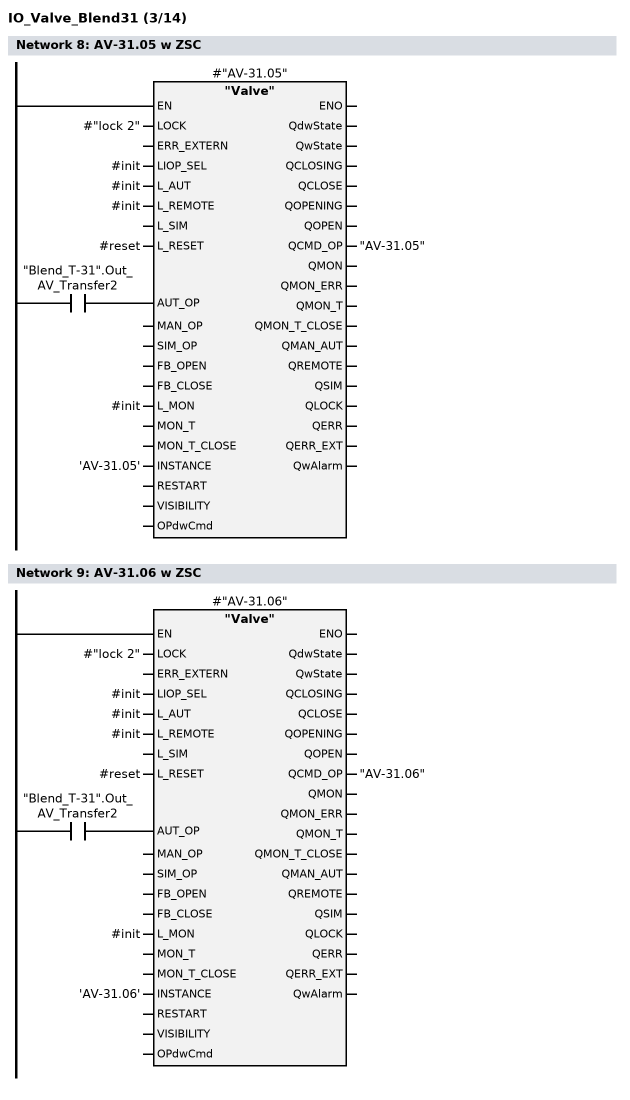
   RUNG wire#powerrail
      #"AV-31.05"(AUT_OP := wire#w1, LOCK := #"lock 2", ERR_EXTERN :=, LIOP_SEL := #init, L_AUT := #init, L_REMOTE := #init, L_SIM :=, L_RESET := #reset, MAN_OP :=, SIM_OP :=, FB_OPEN :=, FB_CLOSE :=, L_MON := #init, MON_T :=, MON_T_CLOSE :=, INSTANCE := 'AV-31.05', RESTART :=, VISIBILITY :=, OPdwCmd :=, QdwState =>, QwState =>, QCLOSING =>, QCLOSE =>, QOPENING =>, QOPEN =>, QCMD_OP => "AV-31.05", QMON =>, QMON_ERR =>, QMON_T =>, QMON_T_CLOSE =>, QMAN_AUT =>, QREMOTE =>, QSIM =>, QLOCK =>, QERR =>, QERR_EXT =>, QwAlarm =>)
   END_RUNG
   RUNG wire#powerrail
      Contact( "Blend_T-31".Out_AV_Transfer2 )
   END_RUNG wire#w1
   // the same network as SCL:
   #"AV-31.05"(LOCK := #"lock 2",   // "Valve"
               LIOP_SEL := #init,
               L_AUT := #init,
               L_REMOTE := #init,
               L_RESET := #reset,
               AUT_OP := "Blend_T-31".Out_AV_Transfer2,
               L_MON := #init,
               INSTANCE := 'AV-31.05',
               QCMD_OP => "AV-31.05");
END_REGION

REGION Network 9: AV-31.06 w ZSC
   RUNG wire#powerrail
      #"AV-31.06"(AUT_OP := wire#w1, LOCK := #"lock 2", ERR_EXTERN :=, LIOP_SEL := #init, L_AUT := #init, L_REMOTE := #init, L_SIM :=, L_RESET := #reset, MAN_OP :=, SIM_OP :=, FB_OPEN :=, FB_CLOSE :=, L_MON := #init, MON_T :=, MON_T_CLOSE :=, INSTANCE := 'AV-31.06', RESTART :=, VISIBILITY :=, OPdwCmd :=, QdwState =>, QwState =>, QCLOSING =>, QCLOSE =>, QOPENING =>, QOPEN =>, QCMD_OP => "AV-31.06", QMON =>, QMON_ERR =>, QMON_T =>, QMON_T_CLOSE =>, QMAN_AUT =>, QREMOTE =>, QSIM =>, QLOCK =>, QERR =>, QERR_EXT =>, QwAlarm =>)
   END_RUNG
   RUNG wire#powerrail
      Contact( "Blend_T-31".Out_AV_Transfer2 )
   END_RUNG wire#w1
   // the same network as SCL:
   #"AV-31.06"(LOCK := #"lock 2",   // "Valve"
               LIOP_SEL := #init,
               L_AUT := #init,
               L_REMOTE := #init,
               L_RESET := #reset,
               AUT_OP := "Blend_T-31".Out_AV_Transfer2,
               L_MON := #init,
               INSTANCE := 'AV-31.06',
               QCMD_OP => "AV-31.06");
END_REGION

REGION Network 10: AV-31.07
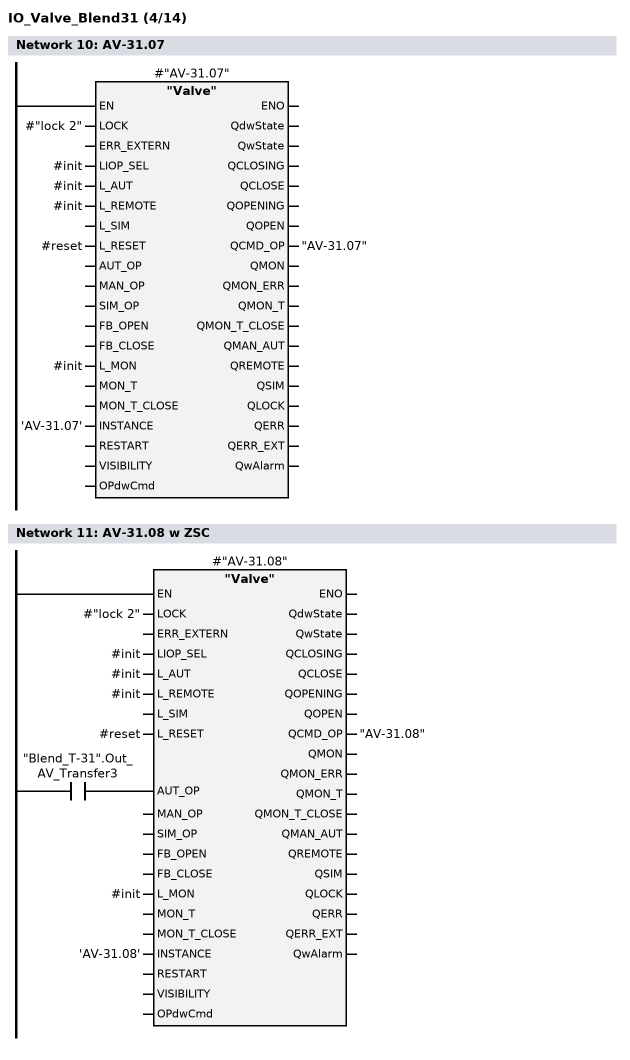
   RUNG wire#powerrail
      #"AV-31.07"(LOCK := #"lock 2", ERR_EXTERN :=, LIOP_SEL := #init, L_AUT := #init, L_REMOTE := #init, L_SIM :=, L_RESET := #reset, AUT_OP :=, MAN_OP :=, SIM_OP :=, FB_OPEN :=, FB_CLOSE :=, L_MON := #init, MON_T :=, MON_T_CLOSE :=, INSTANCE := 'AV-31.07', RESTART :=, VISIBILITY :=, OPdwCmd :=, QdwState =>, QwState =>, QCLOSING =>, QCLOSE =>, QOPENING =>, QOPEN =>, QCMD_OP => "AV-31.07", QMON =>, QMON_ERR =>, QMON_T =>, QMON_T_CLOSE =>, QMAN_AUT =>, QREMOTE =>, QSIM =>, QLOCK =>, QERR =>, QERR_EXT =>, QwAlarm =>)
   END_RUNG
   // the same network as SCL:
   #"AV-31.07"(LOCK := #"lock 2",   // "Valve"
               LIOP_SEL := #init,
               L_AUT := #init,
               L_REMOTE := #init,
               L_RESET := #reset,
               L_MON := #init,
               INSTANCE := 'AV-31.07',
               QCMD_OP => "AV-31.07");
END_REGION

REGION Network 11: AV-31.08 w ZSC
   RUNG wire#powerrail
      #"AV-31.08"(AUT_OP := wire#w1, LOCK := #"lock 2", ERR_EXTERN :=, LIOP_SEL := #init, L_AUT := #init, L_REMOTE := #init, L_SIM :=, L_RESET := #reset, MAN_OP :=, SIM_OP :=, FB_OPEN :=, FB_CLOSE :=, L_MON := #init, MON_T :=, MON_T_CLOSE :=, INSTANCE := 'AV-31.08', RESTART :=, VISIBILITY :=, OPdwCmd :=, QdwState =>, QwState =>, QCLOSING =>, QCLOSE =>, QOPENING =>, QOPEN =>, QCMD_OP => "AV-31.08", QMON =>, QMON_ERR =>, QMON_T =>, QMON_T_CLOSE =>, QMAN_AUT =>, QREMOTE =>, QSIM =>, QLOCK =>, QERR =>, QERR_EXT =>, QwAlarm =>)
   END_RUNG
   RUNG wire#powerrail
      Contact( "Blend_T-31".Out_AV_Transfer3 )
   END_RUNG wire#w1
   // the same network as SCL:
   #"AV-31.08"(LOCK := #"lock 2",   // "Valve"
               LIOP_SEL := #init,
               L_AUT := #init,
               L_REMOTE := #init,
               L_RESET := #reset,
               AUT_OP := "Blend_T-31".Out_AV_Transfer3,
               L_MON := #init,
               INSTANCE := 'AV-31.08',
               QCMD_OP => "AV-31.08");
END_REGION

REGION Network 12: AV-31.09 w ZSC
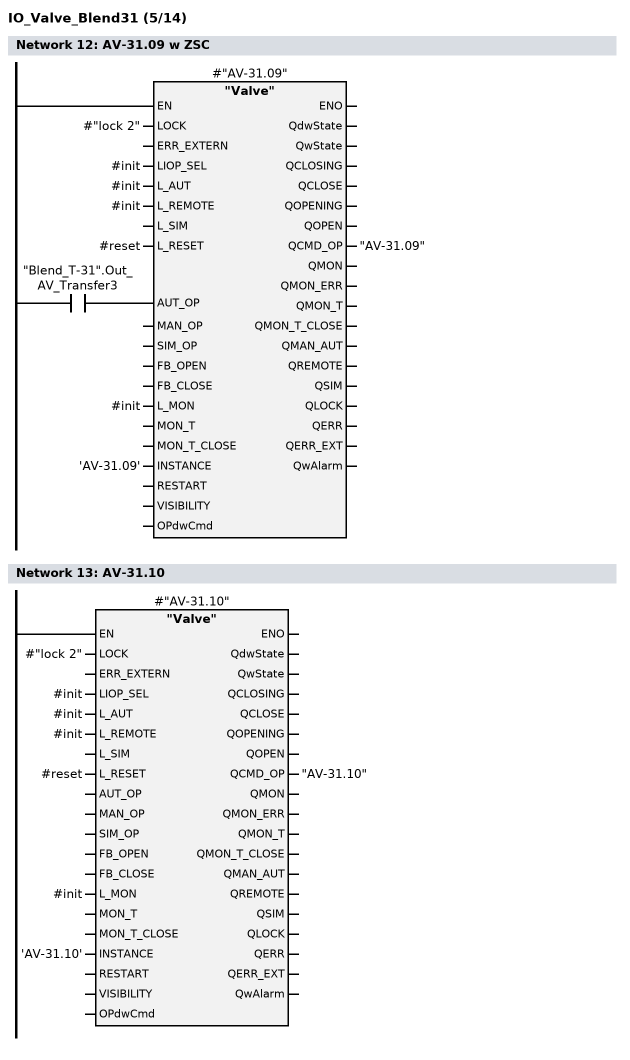
   RUNG wire#powerrail
      #"AV-31.09"(AUT_OP := wire#w1, LOCK := #"lock 2", ERR_EXTERN :=, LIOP_SEL := #init, L_AUT := #init, L_REMOTE := #init, L_SIM :=, L_RESET := #reset, MAN_OP :=, SIM_OP :=, FB_OPEN :=, FB_CLOSE :=, L_MON := #init, MON_T :=, MON_T_CLOSE :=, INSTANCE := 'AV-31.09', RESTART :=, VISIBILITY :=, OPdwCmd :=, QdwState =>, QwState =>, QCLOSING =>, QCLOSE =>, QOPENING =>, QOPEN =>, QCMD_OP => "AV-31.09", QMON =>, QMON_ERR =>, QMON_T =>, QMON_T_CLOSE =>, QMAN_AUT =>, QREMOTE =>, QSIM =>, QLOCK =>, QERR =>, QERR_EXT =>, QwAlarm =>)
   END_RUNG
   RUNG wire#powerrail
      Contact( "Blend_T-31".Out_AV_Transfer3 )
   END_RUNG wire#w1
   // the same network as SCL:
   #"AV-31.09"(LOCK := #"lock 2",   // "Valve"
               LIOP_SEL := #init,
               L_AUT := #init,
               L_REMOTE := #init,
               L_RESET := #reset,
               AUT_OP := "Blend_T-31".Out_AV_Transfer3,
               L_MON := #init,
               INSTANCE := 'AV-31.09',
               QCMD_OP => "AV-31.09");
END_REGION

REGION Network 13: AV-31.10
   RUNG wire#powerrail
      #"AV-31.10"(LOCK := #"lock 2", ERR_EXTERN :=, LIOP_SEL := #init, L_AUT := #init, L_REMOTE := #init, L_SIM :=, L_RESET := #reset, AUT_OP :=, MAN_OP :=, SIM_OP :=, FB_OPEN :=, FB_CLOSE :=, L_MON := #init, MON_T :=, MON_T_CLOSE :=, INSTANCE := 'AV-31.10', RESTART :=, VISIBILITY :=, OPdwCmd :=, QdwState =>, QwState =>, QCLOSING =>, QCLOSE =>, QOPENING =>, QOPEN =>, QCMD_OP => "AV-31.10", QMON =>, QMON_ERR =>, QMON_T =>, QMON_T_CLOSE =>, QMAN_AUT =>, QREMOTE =>, QSIM =>, QLOCK =>, QERR =>, QERR_EXT =>, QwAlarm =>)
   END_RUNG
   // the same network as SCL:
   #"AV-31.10"(LOCK := #"lock 2",   // "Valve"
               LIOP_SEL := #init,
               L_AUT := #init,
               L_REMOTE := #init,
               L_RESET := #reset,
               L_MON := #init,
               INSTANCE := 'AV-31.10',
               QCMD_OP => "AV-31.10");
END_REGION

REGION Network 14: AV-31.11 w ZSC
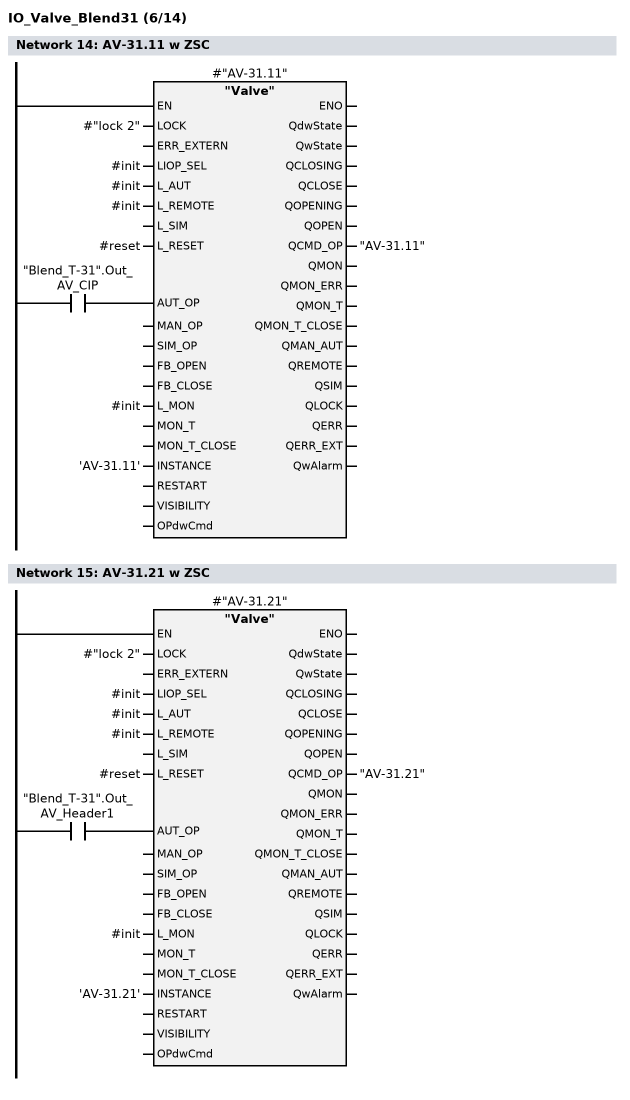
   RUNG wire#powerrail
      #"AV-31.11"(AUT_OP := wire#w1, LOCK := #"lock 2", ERR_EXTERN :=, LIOP_SEL := #init, L_AUT := #init, L_REMOTE := #init, L_SIM :=, L_RESET := #reset, MAN_OP :=, SIM_OP :=, FB_OPEN :=, FB_CLOSE :=, L_MON := #init, MON_T :=, MON_T_CLOSE :=, INSTANCE := 'AV-31.11', RESTART :=, VISIBILITY :=, OPdwCmd :=, QdwState =>, QwState =>, QCLOSING =>, QCLOSE =>, QOPENING =>, QOPEN =>, QCMD_OP => "AV-31.11", QMON =>, QMON_ERR =>, QMON_T =>, QMON_T_CLOSE =>, QMAN_AUT =>, QREMOTE =>, QSIM =>, QLOCK =>, QERR =>, QERR_EXT =>, QwAlarm =>)
   END_RUNG
   RUNG wire#powerrail
      Contact( "Blend_T-31".Out_AV_CIP )
   END_RUNG wire#w1
   // the same network as SCL:
   #"AV-31.11"(LOCK := #"lock 2",   // "Valve"
               LIOP_SEL := #init,
               L_AUT := #init,
               L_REMOTE := #init,
               L_RESET := #reset,
               AUT_OP := "Blend_T-31".Out_AV_CIP,
               L_MON := #init,
               INSTANCE := 'AV-31.11',
               QCMD_OP => "AV-31.11");
END_REGION

REGION Network 15: AV-31.21 w ZSC
   RUNG wire#powerrail
      #"AV-31.21"(AUT_OP := wire#w1, LOCK := #"lock 2", ERR_EXTERN :=, LIOP_SEL := #init, L_AUT := #init, L_REMOTE := #init, L_SIM :=, L_RESET := #reset, MAN_OP :=, SIM_OP :=, FB_OPEN :=, FB_CLOSE :=, L_MON := #init, MON_T :=, MON_T_CLOSE :=, INSTANCE := 'AV-31.21', RESTART :=, VISIBILITY :=, OPdwCmd :=, QdwState =>, QwState =>, QCLOSING =>, QCLOSE =>, QOPENING =>, QOPEN =>, QCMD_OP => "AV-31.21", QMON =>, QMON_ERR =>, QMON_T =>, QMON_T_CLOSE =>, QMAN_AUT =>, QREMOTE =>, QSIM =>, QLOCK =>, QERR =>, QERR_EXT =>, QwAlarm =>)
   END_RUNG
   RUNG wire#powerrail
      Contact( "Blend_T-31".Out_AV_Header1 )
   END_RUNG wire#w1
   // the same network as SCL:
   #"AV-31.21"(LOCK := #"lock 2",   // "Valve"
               LIOP_SEL := #init,
               L_AUT := #init,
               L_REMOTE := #init,
               L_RESET := #reset,
               AUT_OP := "Blend_T-31".Out_AV_Header1,
               L_MON := #init,
               INSTANCE := 'AV-31.21',
               QCMD_OP => "AV-31.21");
END_REGION

REGION Network 16: AV-31.22
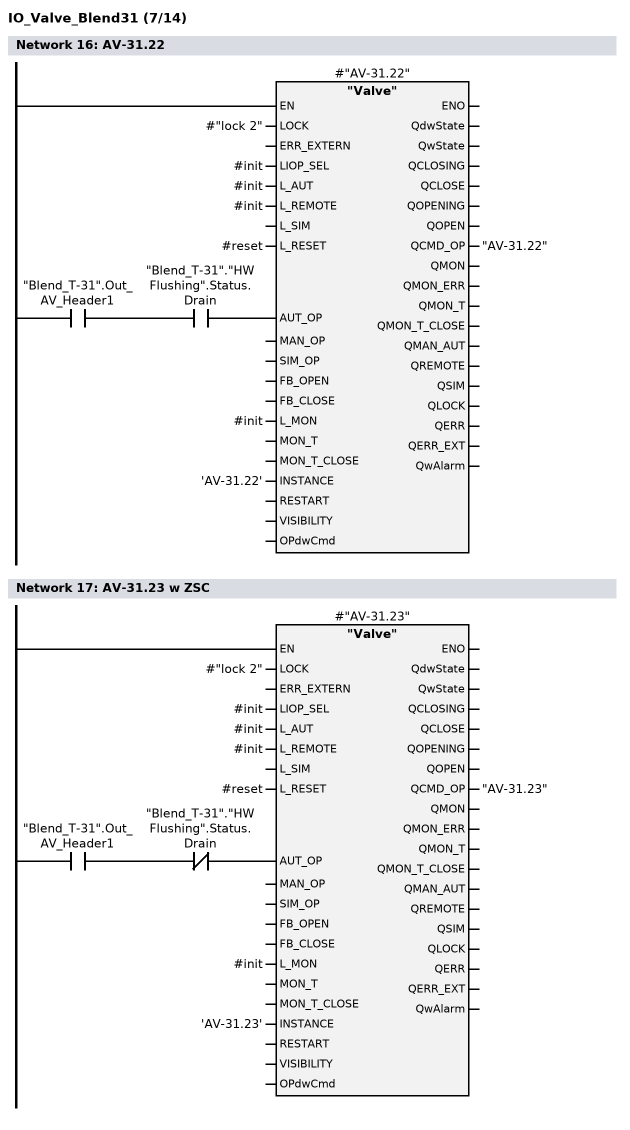
   RUNG wire#powerrail
      #"AV-31.22"(AUT_OP := wire#w1, LOCK := #"lock 2", ERR_EXTERN :=, LIOP_SEL := #init, L_AUT := #init, L_REMOTE := #init, L_SIM :=, L_RESET := #reset, MAN_OP :=, SIM_OP :=, FB_OPEN :=, FB_CLOSE :=, L_MON := #init, MON_T :=, MON_T_CLOSE :=, INSTANCE := 'AV-31.22', RESTART :=, VISIBILITY :=, OPdwCmd :=, QdwState =>, QwState =>, QCLOSING =>, QCLOSE =>, QOPENING =>, QOPEN =>, QCMD_OP => "AV-31.22", QMON =>, QMON_ERR =>, QMON_T =>, QMON_T_CLOSE =>, QMAN_AUT =>, QREMOTE =>, QSIM =>, QLOCK =>, QERR =>, QERR_EXT =>, QwAlarm =>)
   END_RUNG
   RUNG wire#powerrail
      Contact( "Blend_T-31".Out_AV_Header1 )
      Contact( "Blend_T-31"."HW Flushing".Status.Drain )
   END_RUNG wire#w1
   // the same network as SCL:
   #"AV-31.22"(LOCK := #"lock 2",   // "Valve"
               LIOP_SEL := #init,
               L_AUT := #init,
               L_REMOTE := #init,
               L_RESET := #reset,
               AUT_OP := "Blend_T-31".Out_AV_Header1 AND "Blend_T-31"."HW Flushing".Status.Drain,
               L_MON := #init,
               INSTANCE := 'AV-31.22',
               QCMD_OP => "AV-31.22");
END_REGION

REGION Network 17: AV-31.23 w ZSC
   RUNG wire#powerrail
      #"AV-31.23"(AUT_OP := wire#w1, LOCK := #"lock 2", ERR_EXTERN :=, LIOP_SEL := #init, L_AUT := #init, L_REMOTE := #init, L_SIM :=, L_RESET := #reset, MAN_OP :=, SIM_OP :=, FB_OPEN :=, FB_CLOSE :=, L_MON := #init, MON_T :=, MON_T_CLOSE :=, INSTANCE := 'AV-31.23', RESTART :=, VISIBILITY :=, OPdwCmd :=, QdwState =>, QwState =>, QCLOSING =>, QCLOSE =>, QOPENING =>, QOPEN =>, QCMD_OP => "AV-31.23", QMON =>, QMON_ERR =>, QMON_T =>, QMON_T_CLOSE =>, QMAN_AUT =>, QREMOTE =>, QSIM =>, QLOCK =>, QERR =>, QERR_EXT =>, QwAlarm =>)
   END_RUNG
   RUNG wire#powerrail
      Contact( "Blend_T-31".Out_AV_Header1 )
      I_Contact( "Blend_T-31"."HW Flushing".Status.Drain )
   END_RUNG wire#w1
   // the same network as SCL:
   #"AV-31.23"(LOCK := #"lock 2",   // "Valve"
               LIOP_SEL := #init,
               L_AUT := #init,
               L_REMOTE := #init,
               L_RESET := #reset,
               AUT_OP := "Blend_T-31".Out_AV_Header1 AND NOT "Blend_T-31"."HW Flushing".Status.Drain,
               L_MON := #init,
               INSTANCE := 'AV-31.23',
               QCMD_OP => "AV-31.23");
END_REGION

REGION Network 18: AV-31.24 w ZSC
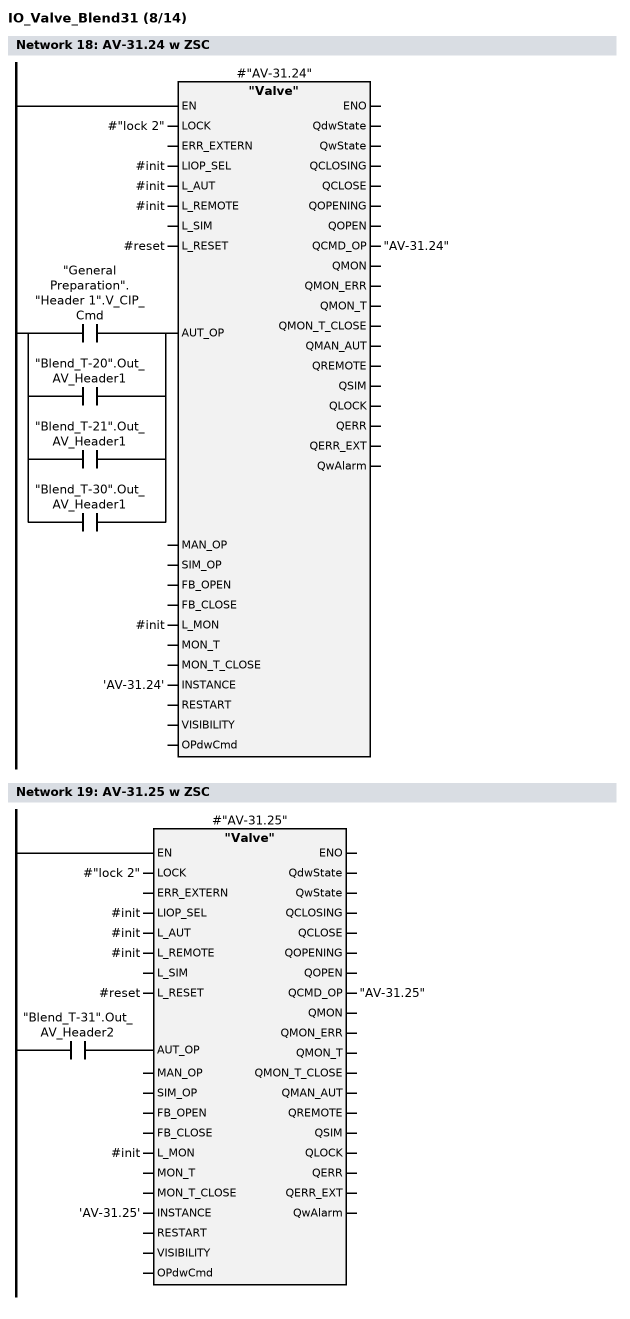
   RUNG wire#powerrail
      #"AV-31.24"(AUT_OP := wire#w1, LOCK := #"lock 2", ERR_EXTERN :=, LIOP_SEL := #init, L_AUT := #init, L_REMOTE := #init, L_SIM :=, L_RESET := #reset, MAN_OP :=, SIM_OP :=, FB_OPEN :=, FB_CLOSE :=, L_MON := #init, MON_T :=, MON_T_CLOSE :=, INSTANCE := 'AV-31.24', RESTART :=, VISIBILITY :=, OPdwCmd :=, QdwState =>, QwState =>, QCLOSING =>, QCLOSE =>, QOPENING =>, QOPEN =>, QCMD_OP => "AV-31.24", QMON =>, QMON_ERR =>, QMON_T =>, QMON_T_CLOSE =>, QMAN_AUT =>, QREMOTE =>, QSIM =>, QLOCK =>, QERR =>, QERR_EXT =>, QwAlarm =>)
   END_RUNG
   RUNG wire#powerrail
      Contact( "General Preparation"."Header 1".V_CIP_Cmd )
   END_RUNG wire#w1
   RUNG wire#powerrail
      Contact( "Blend_T-20".Out_AV_Header1 )
   END_RUNG wire#w1
   RUNG wire#powerrail
      Contact( "Blend_T-21".Out_AV_Header1 )
   END_RUNG wire#w1
   RUNG wire#powerrail
      Contact( "Blend_T-30".Out_AV_Header1 )
   END_RUNG wire#w1
   // the same network as SCL:
   #"AV-31.24"(LOCK := #"lock 2",   // "Valve"
               LIOP_SEL := #init,
               L_AUT := #init,
               L_REMOTE := #init,
               L_RESET := #reset,
               AUT_OP := "General Preparation"."Header 1".V_CIP_Cmd OR "Blend_T-20".Out_AV_Header1 OR "Blend_T-21".Out_AV_Header1 OR "Blend_T-30".Out_AV_Header1,
               L_MON := #init,
               INSTANCE := 'AV-31.24',
               QCMD_OP => "AV-31.24");
END_REGION

REGION Network 19: AV-31.25 w ZSC
   RUNG wire#powerrail
      #"AV-31.25"(AUT_OP := wire#w1, LOCK := #"lock 2", ERR_EXTERN :=, LIOP_SEL := #init, L_AUT := #init, L_REMOTE := #init, L_SIM :=, L_RESET := #reset, MAN_OP :=, SIM_OP :=, FB_OPEN :=, FB_CLOSE :=, L_MON := #init, MON_T :=, MON_T_CLOSE :=, INSTANCE := 'AV-31.25', RESTART :=, VISIBILITY :=, OPdwCmd :=, QdwState =>, QwState =>, QCLOSING =>, QCLOSE =>, QOPENING =>, QOPEN =>, QCMD_OP => "AV-31.25", QMON =>, QMON_ERR =>, QMON_T =>, QMON_T_CLOSE =>, QMAN_AUT =>, QREMOTE =>, QSIM =>, QLOCK =>, QERR =>, QERR_EXT =>, QwAlarm =>)
   END_RUNG
   RUNG wire#powerrail
      Contact( "Blend_T-31".Out_AV_Header2 )
   END_RUNG wire#w1
   // the same network as SCL:
   #"AV-31.25"(LOCK := #"lock 2",   // "Valve"
               LIOP_SEL := #init,
               L_AUT := #init,
               L_REMOTE := #init,
               L_RESET := #reset,
               AUT_OP := "Blend_T-31".Out_AV_Header2,
               L_MON := #init,
               INSTANCE := 'AV-31.25',
               QCMD_OP => "AV-31.25");
END_REGION

REGION Network 20: AV-31.26
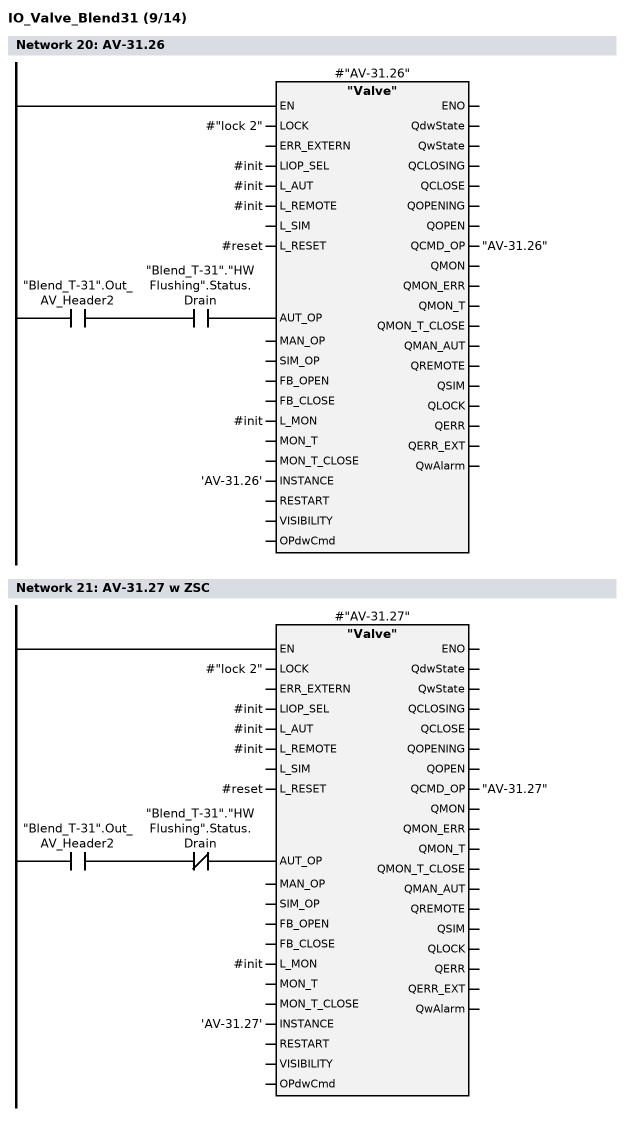
   RUNG wire#powerrail
      #"AV-31.26"(AUT_OP := wire#w1, LOCK := #"lock 2", ERR_EXTERN :=, LIOP_SEL := #init, L_AUT := #init, L_REMOTE := #init, L_SIM :=, L_RESET := #reset, MAN_OP :=, SIM_OP :=, FB_OPEN :=, FB_CLOSE :=, L_MON := #init, MON_T :=, MON_T_CLOSE :=, INSTANCE := 'AV-31.26', RESTART :=, VISIBILITY :=, OPdwCmd :=, QdwState =>, QwState =>, QCLOSING =>, QCLOSE =>, QOPENING =>, QOPEN =>, QCMD_OP => "AV-31.26", QMON =>, QMON_ERR =>, QMON_T =>, QMON_T_CLOSE =>, QMAN_AUT =>, QREMOTE =>, QSIM =>, QLOCK =>, QERR =>, QERR_EXT =>, QwAlarm =>)
   END_RUNG
   RUNG wire#powerrail
      Contact( "Blend_T-31".Out_AV_Header2 )
      Contact( "Blend_T-31"."HW Flushing".Status.Drain )
   END_RUNG wire#w1
   // the same network as SCL:
   #"AV-31.26"(LOCK := #"lock 2",   // "Valve"
               LIOP_SEL := #init,
               L_AUT := #init,
               L_REMOTE := #init,
               L_RESET := #reset,
               AUT_OP := "Blend_T-31".Out_AV_Header2 AND "Blend_T-31"."HW Flushing".Status.Drain,
               L_MON := #init,
               INSTANCE := 'AV-31.26',
               QCMD_OP => "AV-31.26");
END_REGION

REGION Network 21: AV-31.27 w ZSC
   RUNG wire#powerrail
      #"AV-31.27"(AUT_OP := wire#w1, LOCK := #"lock 2", ERR_EXTERN :=, LIOP_SEL := #init, L_AUT := #init, L_REMOTE := #init, L_SIM :=, L_RESET := #reset, MAN_OP :=, SIM_OP :=, FB_OPEN :=, FB_CLOSE :=, L_MON := #init, MON_T :=, MON_T_CLOSE :=, INSTANCE := 'AV-31.27', RESTART :=, VISIBILITY :=, OPdwCmd :=, QdwState =>, QwState =>, QCLOSING =>, QCLOSE =>, QOPENING =>, QOPEN =>, QCMD_OP => "AV-31.27", QMON =>, QMON_ERR =>, QMON_T =>, QMON_T_CLOSE =>, QMAN_AUT =>, QREMOTE =>, QSIM =>, QLOCK =>, QERR =>, QERR_EXT =>, QwAlarm =>)
   END_RUNG
   RUNG wire#powerrail
      Contact( "Blend_T-31".Out_AV_Header2 )
      I_Contact( "Blend_T-31"."HW Flushing".Status.Drain )
   END_RUNG wire#w1
   // the same network as SCL:
   #"AV-31.27"(LOCK := #"lock 2",   // "Valve"
               LIOP_SEL := #init,
               L_AUT := #init,
               L_REMOTE := #init,
               L_RESET := #reset,
               AUT_OP := "Blend_T-31".Out_AV_Header2 AND NOT "Blend_T-31"."HW Flushing".Status.Drain,
               L_MON := #init,
               INSTANCE := 'AV-31.27',
               QCMD_OP => "AV-31.27");
END_REGION

REGION Network 22: AV-31.28 w ZSC
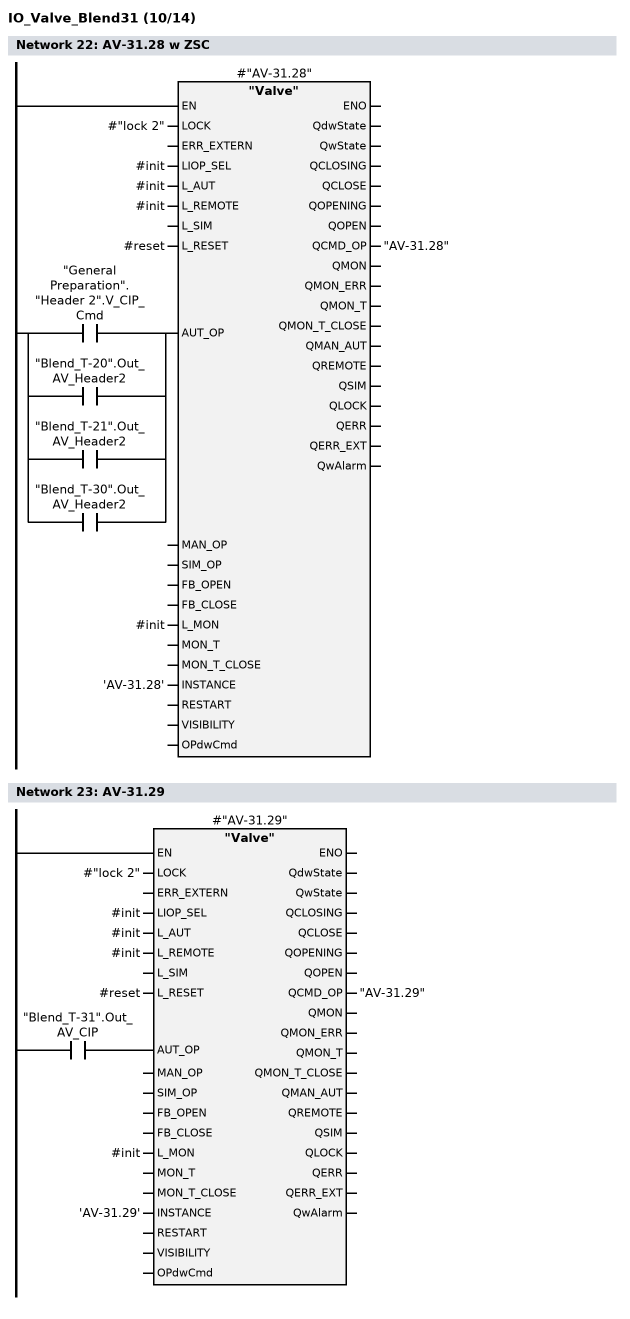
   RUNG wire#powerrail
      #"AV-31.28"(AUT_OP := wire#w1, LOCK := #"lock 2", ERR_EXTERN :=, LIOP_SEL := #init, L_AUT := #init, L_REMOTE := #init, L_SIM :=, L_RESET := #reset, MAN_OP :=, SIM_OP :=, FB_OPEN :=, FB_CLOSE :=, L_MON := #init, MON_T :=, MON_T_CLOSE :=, INSTANCE := 'AV-31.28', RESTART :=, VISIBILITY :=, OPdwCmd :=, QdwState =>, QwState =>, QCLOSING =>, QCLOSE =>, QOPENING =>, QOPEN =>, QCMD_OP => "AV-31.28", QMON =>, QMON_ERR =>, QMON_T =>, QMON_T_CLOSE =>, QMAN_AUT =>, QREMOTE =>, QSIM =>, QLOCK =>, QERR =>, QERR_EXT =>, QwAlarm =>)
   END_RUNG
   RUNG wire#powerrail
      Contact( "General Preparation"."Header 2".V_CIP_Cmd )
   END_RUNG wire#w1
   RUNG wire#powerrail
      Contact( "Blend_T-20".Out_AV_Header2 )
   END_RUNG wire#w1
   RUNG wire#powerrail
      Contact( "Blend_T-21".Out_AV_Header2 )
   END_RUNG wire#w1
   RUNG wire#powerrail
      Contact( "Blend_T-30".Out_AV_Header2 )
   END_RUNG wire#w1
   // the same network as SCL:
   #"AV-31.28"(LOCK := #"lock 2",   // "Valve"
               LIOP_SEL := #init,
               L_AUT := #init,
               L_REMOTE := #init,
               L_RESET := #reset,
               AUT_OP := "General Preparation"."Header 2".V_CIP_Cmd OR "Blend_T-20".Out_AV_Header2 OR "Blend_T-21".Out_AV_Header2 OR "Blend_T-30".Out_AV_Header2,
               L_MON := #init,
               INSTANCE := 'AV-31.28',
               QCMD_OP => "AV-31.28");
END_REGION

REGION Network 23: AV-31.29
   RUNG wire#powerrail
      #"AV-31.29"(AUT_OP := wire#w1, LOCK := #"lock 2", ERR_EXTERN :=, LIOP_SEL := #init, L_AUT := #init, L_REMOTE := #init, L_SIM :=, L_RESET := #reset, MAN_OP :=, SIM_OP :=, FB_OPEN :=, FB_CLOSE :=, L_MON := #init, MON_T :=, MON_T_CLOSE :=, INSTANCE := 'AV-31.29', RESTART :=, VISIBILITY :=, OPdwCmd :=, QdwState =>, QwState =>, QCLOSING =>, QCLOSE =>, QOPENING =>, QOPEN =>, QCMD_OP => "AV-31.29", QMON =>, QMON_ERR =>, QMON_T =>, QMON_T_CLOSE =>, QMAN_AUT =>, QREMOTE =>, QSIM =>, QLOCK =>, QERR =>, QERR_EXT =>, QwAlarm =>)
   END_RUNG
   RUNG wire#powerrail
      Contact( "Blend_T-31".Out_AV_CIP )
   END_RUNG wire#w1
   // the same network as SCL:
   #"AV-31.29"(LOCK := #"lock 2",   // "Valve"
               LIOP_SEL := #init,
               L_AUT := #init,
               L_REMOTE := #init,
               L_RESET := #reset,
               AUT_OP := "Blend_T-31".Out_AV_CIP,
               L_MON := #init,
               INSTANCE := 'AV-31.29',
               QCMD_OP => "AV-31.29");
END_REGION

REGION Network 24: AV-31.30
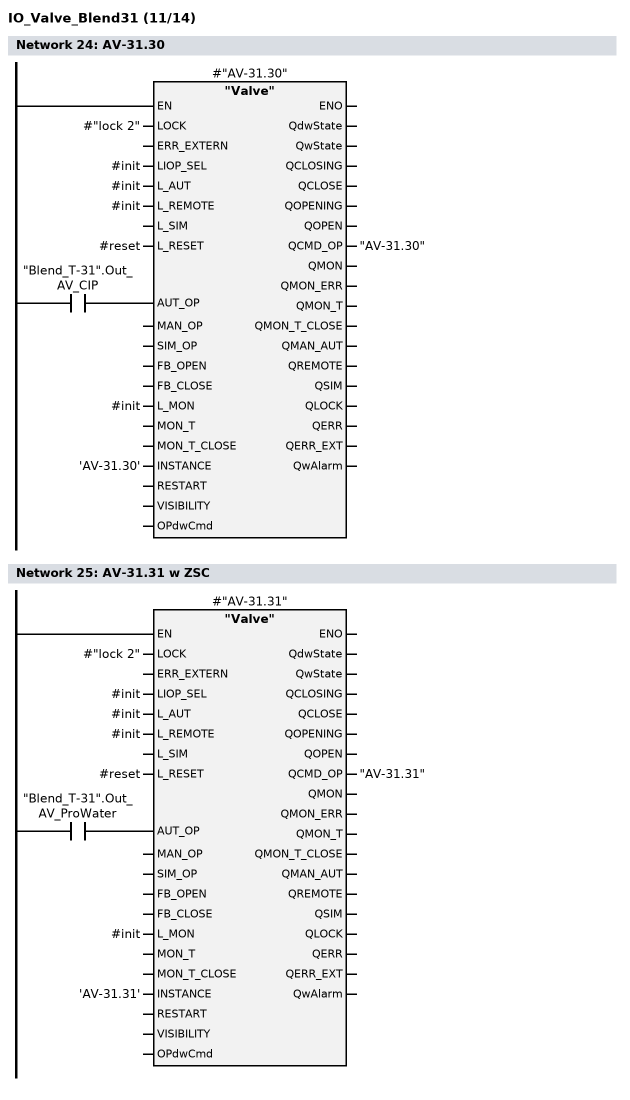
   RUNG wire#powerrail
      #"AV-31.30"(AUT_OP := wire#w1, LOCK := #"lock 2", ERR_EXTERN :=, LIOP_SEL := #init, L_AUT := #init, L_REMOTE := #init, L_SIM :=, L_RESET := #reset, MAN_OP :=, SIM_OP :=, FB_OPEN :=, FB_CLOSE :=, L_MON := #init, MON_T :=, MON_T_CLOSE :=, INSTANCE := 'AV-31.30', RESTART :=, VISIBILITY :=, OPdwCmd :=, QdwState =>, QwState =>, QCLOSING =>, QCLOSE =>, QOPENING =>, QOPEN =>, QCMD_OP => "AV-31.30", QMON =>, QMON_ERR =>, QMON_T =>, QMON_T_CLOSE =>, QMAN_AUT =>, QREMOTE =>, QSIM =>, QLOCK =>, QERR =>, QERR_EXT =>, QwAlarm =>)
   END_RUNG
   RUNG wire#powerrail
      Contact( "Blend_T-31".Out_AV_CIP )
   END_RUNG wire#w1
   // the same network as SCL:
   #"AV-31.30"(LOCK := #"lock 2",   // "Valve"
               LIOP_SEL := #init,
               L_AUT := #init,
               L_REMOTE := #init,
               L_RESET := #reset,
               AUT_OP := "Blend_T-31".Out_AV_CIP,
               L_MON := #init,
               INSTANCE := 'AV-31.30',
               QCMD_OP => "AV-31.30");
END_REGION

REGION Network 25: AV-31.31 w ZSC
   RUNG wire#powerrail
      #"AV-31.31"(AUT_OP := wire#w1, LOCK := #"lock 2", ERR_EXTERN :=, LIOP_SEL := #init, L_AUT := #init, L_REMOTE := #init, L_SIM :=, L_RESET := #reset, MAN_OP :=, SIM_OP :=, FB_OPEN :=, FB_CLOSE :=, L_MON := #init, MON_T :=, MON_T_CLOSE :=, INSTANCE := 'AV-31.31', RESTART :=, VISIBILITY :=, OPdwCmd :=, QdwState =>, QwState =>, QCLOSING =>, QCLOSE =>, QOPENING =>, QOPEN =>, QCMD_OP => "AV-31.31", QMON =>, QMON_ERR =>, QMON_T =>, QMON_T_CLOSE =>, QMAN_AUT =>, QREMOTE =>, QSIM =>, QLOCK =>, QERR =>, QERR_EXT =>, QwAlarm =>)
   END_RUNG
   RUNG wire#powerrail
      Contact( "Blend_T-31".Out_AV_ProWater )
   END_RUNG wire#w1
   // the same network as SCL:
   #"AV-31.31"(LOCK := #"lock 2",   // "Valve"
               LIOP_SEL := #init,
               L_AUT := #init,
               L_REMOTE := #init,
               L_RESET := #reset,
               AUT_OP := "Blend_T-31".Out_AV_ProWater,
               L_MON := #init,
               INSTANCE := 'AV-31.31',
               QCMD_OP => "AV-31.31");
END_REGION

REGION Network 26: AV-31.32 w ZSC
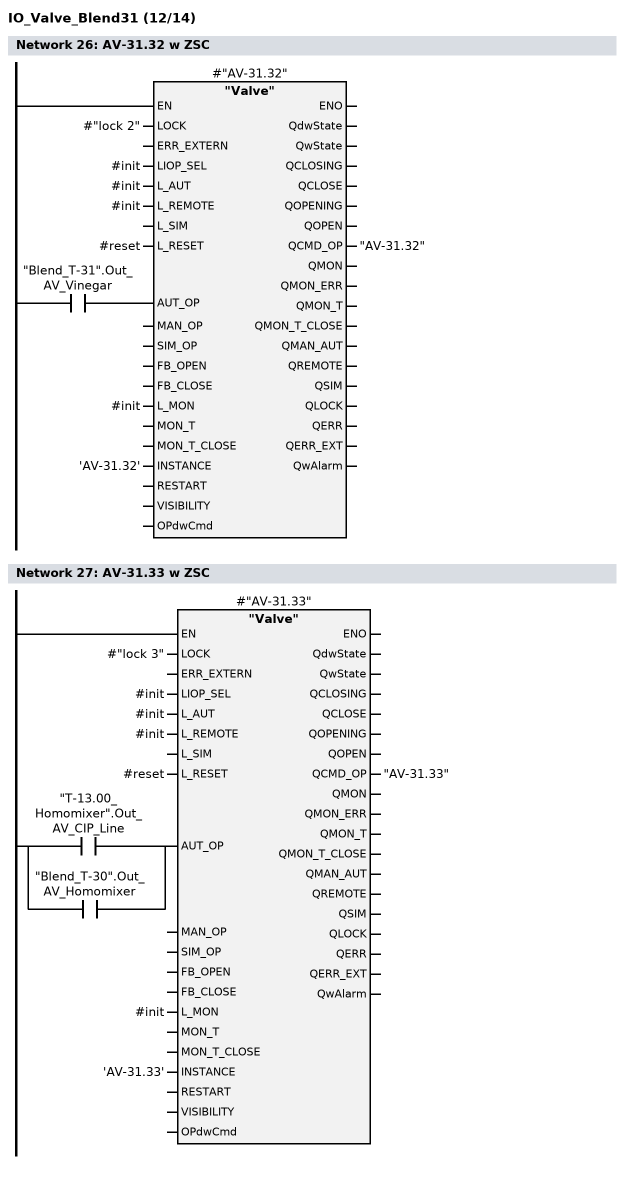
   RUNG wire#powerrail
      #"AV-31.32"(AUT_OP := wire#w1, LOCK := #"lock 2", ERR_EXTERN :=, LIOP_SEL := #init, L_AUT := #init, L_REMOTE := #init, L_SIM :=, L_RESET := #reset, MAN_OP :=, SIM_OP :=, FB_OPEN :=, FB_CLOSE :=, L_MON := #init, MON_T :=, MON_T_CLOSE :=, INSTANCE := 'AV-31.32', RESTART :=, VISIBILITY :=, OPdwCmd :=, QdwState =>, QwState =>, QCLOSING =>, QCLOSE =>, QOPENING =>, QOPEN =>, QCMD_OP => "AV-31.32", QMON =>, QMON_ERR =>, QMON_T =>, QMON_T_CLOSE =>, QMAN_AUT =>, QREMOTE =>, QSIM =>, QLOCK =>, QERR =>, QERR_EXT =>, QwAlarm =>)
   END_RUNG
   RUNG wire#powerrail
      Contact( "Blend_T-31".Out_AV_Vinegar )
   END_RUNG wire#w1
   // the same network as SCL:
   #"AV-31.32"(LOCK := #"lock 2",   // "Valve"
               LIOP_SEL := #init,
               L_AUT := #init,
               L_REMOTE := #init,
               L_RESET := #reset,
               AUT_OP := "Blend_T-31".Out_AV_Vinegar,
               L_MON := #init,
               INSTANCE := 'AV-31.32',
               QCMD_OP => "AV-31.32");
END_REGION

REGION Network 27: AV-31.33 w ZSC
   RUNG wire#powerrail
      #"AV-31.33"(AUT_OP := wire#w1, LOCK := #"lock 3", ERR_EXTERN :=, LIOP_SEL := #init, L_AUT := #init, L_REMOTE := #init, L_SIM :=, L_RESET := #reset, MAN_OP :=, SIM_OP :=, FB_OPEN :=, FB_CLOSE :=, L_MON := #init, MON_T :=, MON_T_CLOSE :=, INSTANCE := 'AV-31.33', RESTART :=, VISIBILITY :=, OPdwCmd :=, QdwState =>, QwState =>, QCLOSING =>, QCLOSE =>, QOPENING =>, QOPEN =>, QCMD_OP => "AV-31.33", QMON =>, QMON_ERR =>, QMON_T =>, QMON_T_CLOSE =>, QMAN_AUT =>, QREMOTE =>, QSIM =>, QLOCK =>, QERR =>, QERR_EXT =>, QwAlarm =>)
   END_RUNG
   RUNG wire#powerrail
      Contact( "T-13.00_Homomixer".Out_AV_CIP_Line )
   END_RUNG wire#w1
   RUNG wire#powerrail
      Contact( "Blend_T-30".Out_AV_Homomixer )
   END_RUNG wire#w1
   // the same network as SCL:
   #"AV-31.33"(LOCK := #"lock 3",   // "Valve"
               LIOP_SEL := #init,
               L_AUT := #init,
               L_REMOTE := #init,
               L_RESET := #reset,
               AUT_OP := "T-13.00_Homomixer".Out_AV_CIP_Line OR "Blend_T-30".Out_AV_Homomixer,
               L_MON := #init,
               INSTANCE := 'AV-31.33',
               QCMD_OP => "AV-31.33");
END_REGION

REGION Network 28: AV-31.34 w ZSC
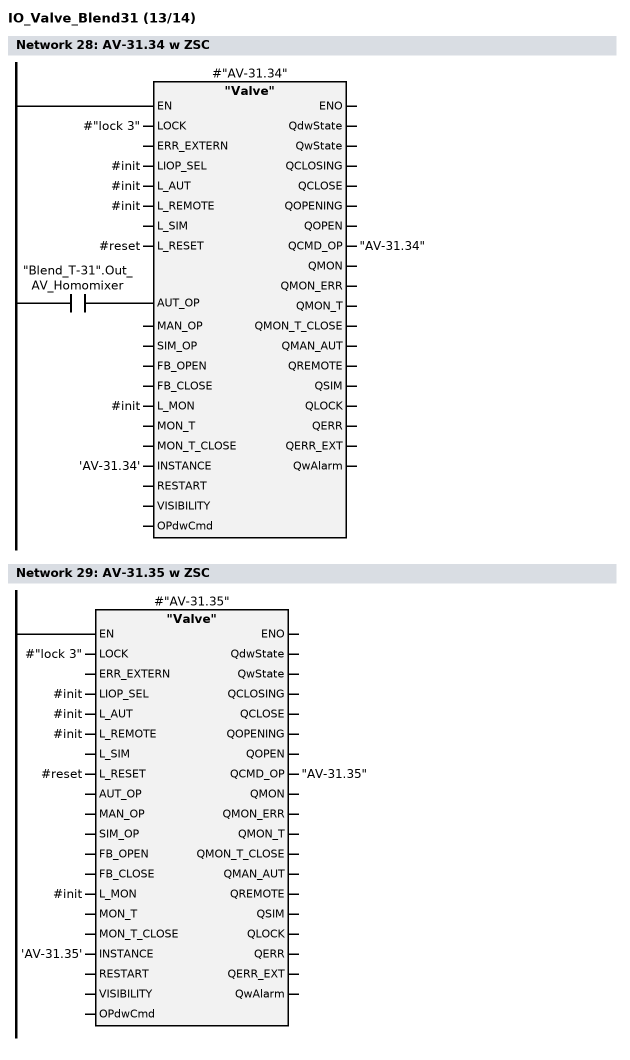
   RUNG wire#powerrail
      #"AV-31.34"(AUT_OP := wire#w1, LOCK := #"lock 3", ERR_EXTERN :=, LIOP_SEL := #init, L_AUT := #init, L_REMOTE := #init, L_SIM :=, L_RESET := #reset, MAN_OP :=, SIM_OP :=, FB_OPEN :=, FB_CLOSE :=, L_MON := #init, MON_T :=, MON_T_CLOSE :=, INSTANCE := 'AV-31.34', RESTART :=, VISIBILITY :=, OPdwCmd :=, QdwState =>, QwState =>, QCLOSING =>, QCLOSE =>, QOPENING =>, QOPEN =>, QCMD_OP => "AV-31.34", QMON =>, QMON_ERR =>, QMON_T =>, QMON_T_CLOSE =>, QMAN_AUT =>, QREMOTE =>, QSIM =>, QLOCK =>, QERR =>, QERR_EXT =>, QwAlarm =>)
   END_RUNG
   RUNG wire#powerrail
      Contact( "Blend_T-31".Out_AV_Homomixer )
   END_RUNG wire#w1
   // the same network as SCL:
   #"AV-31.34"(LOCK := #"lock 3",   // "Valve"
               LIOP_SEL := #init,
               L_AUT := #init,
               L_REMOTE := #init,
               L_RESET := #reset,
               AUT_OP := "Blend_T-31".Out_AV_Homomixer,
               L_MON := #init,
               INSTANCE := 'AV-31.34',
               QCMD_OP => "AV-31.34");
END_REGION

REGION Network 29: AV-31.35 w ZSC
   RUNG wire#powerrail
      #"AV-31.35"(LOCK := #"lock 3", ERR_EXTERN :=, LIOP_SEL := #init, L_AUT := #init, L_REMOTE := #init, L_SIM :=, L_RESET := #reset, AUT_OP :=, MAN_OP :=, SIM_OP :=, FB_OPEN :=, FB_CLOSE :=, L_MON := #init, MON_T :=, MON_T_CLOSE :=, INSTANCE := 'AV-31.35', RESTART :=, VISIBILITY :=, OPdwCmd :=, QdwState =>, QwState =>, QCLOSING =>, QCLOSE =>, QOPENING =>, QOPEN =>, QCMD_OP => "AV-31.35", QMON =>, QMON_ERR =>, QMON_T =>, QMON_T_CLOSE =>, QMAN_AUT =>, QREMOTE =>, QSIM =>, QLOCK =>, QERR =>, QERR_EXT =>, QwAlarm =>)
   END_RUNG
   // the same network as SCL:
   #"AV-31.35"(LOCK := #"lock 3",   // "Valve"
               LIOP_SEL := #init,
               L_AUT := #init,
               L_REMOTE := #init,
               L_RESET := #reset,
               L_MON := #init,
               INSTANCE := 'AV-31.35',
               QCMD_OP => "AV-31.35");
END_REGION

REGION Network 30: AV-31.41
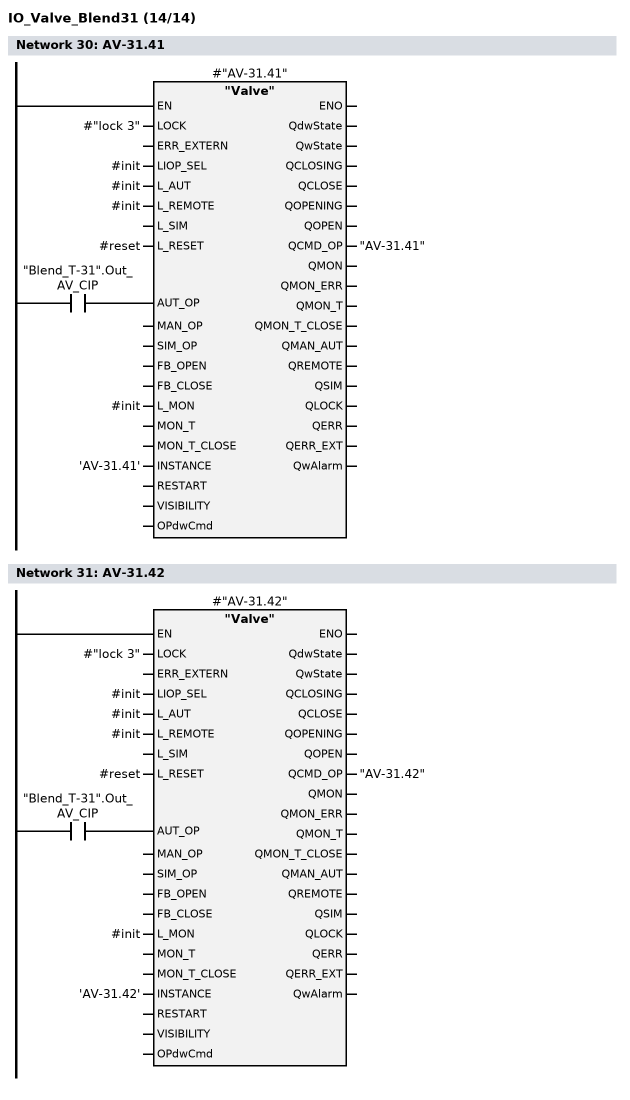
   RUNG wire#powerrail
      #"AV-31.41"(AUT_OP := wire#w1, LOCK := #"lock 3", ERR_EXTERN :=, LIOP_SEL := #init, L_AUT := #init, L_REMOTE := #init, L_SIM :=, L_RESET := #reset, MAN_OP :=, SIM_OP :=, FB_OPEN :=, FB_CLOSE :=, L_MON := #init, MON_T :=, MON_T_CLOSE :=, INSTANCE := 'AV-31.41', RESTART :=, VISIBILITY :=, OPdwCmd :=, QdwState =>, QwState =>, QCLOSING =>, QCLOSE =>, QOPENING =>, QOPEN =>, QCMD_OP => "AV-31.41", QMON =>, QMON_ERR =>, QMON_T =>, QMON_T_CLOSE =>, QMAN_AUT =>, QREMOTE =>, QSIM =>, QLOCK =>, QERR =>, QERR_EXT =>, QwAlarm =>)
   END_RUNG
   RUNG wire#powerrail
      Contact( "Blend_T-31".Out_AV_CIP )
   END_RUNG wire#w1
   // the same network as SCL:
   #"AV-31.41"(LOCK := #"lock 3",   // "Valve"
               LIOP_SEL := #init,
               L_AUT := #init,
               L_REMOTE := #init,
               L_RESET := #reset,
               AUT_OP := "Blend_T-31".Out_AV_CIP,
               L_MON := #init,
               INSTANCE := 'AV-31.41',
               QCMD_OP => "AV-31.41");
END_REGION

REGION Network 31: AV-31.42
   RUNG wire#powerrail
      #"AV-31.42"(AUT_OP := wire#w1, LOCK := #"lock 3", ERR_EXTERN :=, LIOP_SEL := #init, L_AUT := #init, L_REMOTE := #init, L_SIM :=, L_RESET := #reset, MAN_OP :=, SIM_OP :=, FB_OPEN :=, FB_CLOSE :=, L_MON := #init, MON_T :=, MON_T_CLOSE :=, INSTANCE := 'AV-31.42', RESTART :=, VISIBILITY :=, OPdwCmd :=, QdwState =>, QwState =>, QCLOSING =>, QCLOSE =>, QOPENING =>, QOPEN =>, QCMD_OP => "AV-31.42", QMON =>, QMON_ERR =>, QMON_T =>, QMON_T_CLOSE =>, QMAN_AUT =>, QREMOTE =>, QSIM =>, QLOCK =>, QERR =>, QERR_EXT =>, QwAlarm =>)
   END_RUNG
   RUNG wire#powerrail
      Contact( "Blend_T-31".Out_AV_CIP )
   END_RUNG wire#w1
   // the same network as SCL:
   #"AV-31.42"(LOCK := #"lock 3",   // "Valve"
               LIOP_SEL := #init,
               L_AUT := #init,
               L_REMOTE := #init,
               L_RESET := #reset,
               AUT_OP := "Blend_T-31".Out_AV_CIP,
               L_MON := #init,
               INSTANCE := 'AV-31.42',
               QCMD_OP => "AV-31.42");
END_REGION
END_FUNCTION_BLOCK

FUNCTION_BLOCK "IO_Valve_Blend40"   // FB28, LAD
{ S7_Optimized_Access := 'FALSE' }
VERSION : 0.1
// stored: AutoNumber true, IsIECCheckEnabled false, SetENOAutomatically false, UDAEnableTagReadback false
   VAR_INPUT
      "lock 1" : Bool;
      "lock 2" : Bool;
      "lock 3" : Bool;
      "lock 4" : Bool;
      init : Bool;
      reset : Bool;
      testing : Bool;
   END_VAR
   VAR
      "AV-40.01" : "Valve";
      "AV-40.02" : "Valve";
      "AV-40.03" : "Valve";
      "AV-40.04" : "Valve";
      "AV-40.05" : "Valve";
      "AV-40.06" : "Valve";
      "AV-40.07" : "Valve";
      "AV-40.08" : "Valve";
      "AV-40.09" : "Valve";
      "AV-40.10" : "Valve";
      "AV-40.11" : "Valve";
      "AV-40.21" : "Valve";
      "AV-40.22" : "Valve";
      "AV-40.23" : "Valve";
      "AV-40.24" : "Valve";
      "AV-40.25" : "Valve";
      "AV-40.26" : "Valve";
      "AV-40.27" : "Valve";
      "AV-40.28" : "Valve";
      "AV-40.29" : "Valve";
      "AV-40.30" : "Valve";
      "AV-40.31" : "Valve";
      "AV-40.32" : "Valve";
      "AV-40.33" : "Valve";
      "AV-40.34" : "Valve";
   END_VAR
BEGIN

REGION Network 2 (SCL): FB OPEN AND CLOSE VALVE T-40
   IF #testing THEN
       // Statement section IF
       #"AV-40.01".FB_OPEN := #"AV-40.01".QCMD_OP;
       #"AV-40.01".FB_CLOSE := NOT #"AV-40.01".QCMD_OP;
       #"AV-40.02".FB_OPEN := #"AV-40.02".QCMD_OP;
       #"AV-40.02".FB_CLOSE := NOT #"AV-40.02".QCMD_OP;
       #"AV-40.03".FB_OPEN := #"AV-40.03".QCMD_OP;
       #"AV-40.03".FB_CLOSE := NOT #"AV-40.03".QCMD_OP;
       #"AV-40.04".FB_OPEN := #"AV-40.04".QCMD_OP;
       #"AV-40.04".FB_CLOSE := NOT #"AV-40.04".QCMD_OP;
       #"AV-40.05".FB_OPEN := #"AV-40.05".QCMD_OP;
       #"AV-40.05".FB_CLOSE := NOT #"AV-40.05".QCMD_OP;
       #"AV-40.06".FB_OPEN := #"AV-40.06".QCMD_OP;
       #"AV-40.06".FB_CLOSE := NOT #"AV-40.06".QCMD_OP;
       #"AV-40.07".FB_OPEN := #"AV-40.07".QCMD_OP;
       #"AV-40.07".FB_CLOSE := NOT #"AV-40.07".QCMD_OP;
       #"AV-40.08".FB_OPEN := #"AV-40.08".QCMD_OP;
       #"AV-40.08".FB_CLOSE := NOT #"AV-40.08".QCMD_OP;
       #"AV-40.09".FB_OPEN := #"AV-40.09".QCMD_OP;
       #"AV-40.09".FB_CLOSE := NOT #"AV-40.09".QCMD_OP;
       #"AV-40.10".FB_OPEN := #"AV-40.10".QCMD_OP;
       #"AV-40.10".FB_CLOSE := NOT #"AV-40.10".QCMD_OP;
       #"AV-40.11".FB_OPEN := #"AV-40.11".QCMD_OP;
       #"AV-40.11".FB_CLOSE := NOT #"AV-40.11".QCMD_OP;
       #"AV-40.21".FB_OPEN := #"AV-40.21".QCMD_OP;
       #"AV-40.21".FB_CLOSE := NOT #"AV-40.21".QCMD_OP;
       #"AV-40.22".FB_OPEN := #"AV-40.22".QCMD_OP;
       #"AV-40.22".FB_CLOSE := NOT #"AV-40.22".QCMD_OP;
       #"AV-40.23".FB_OPEN := #"AV-40.23".QCMD_OP;
       #"AV-40.23".FB_CLOSE := NOT #"AV-40.23".QCMD_OP;
       #"AV-40.24".FB_OPEN := #"AV-40.24".QCMD_OP;
       #"AV-40.24".FB_CLOSE := NOT #"AV-40.24".QCMD_OP;
       #"AV-40.25".FB_OPEN := #"AV-40.25".QCMD_OP;
       #"AV-40.25".FB_CLOSE := NOT #"AV-40.25".QCMD_OP;
       #"AV-40.26".FB_OPEN := #"AV-40.26".QCMD_OP;
       #"AV-40.26".FB_CLOSE := NOT #"AV-40.26".QCMD_OP;
       #"AV-40.27".FB_OPEN := #"AV-40.27".QCMD_OP;
       #"AV-40.27".FB_CLOSE := NOT #"AV-40.27".QCMD_OP;
       #"AV-40.28".FB_OPEN := #"AV-40.28".QCMD_OP;
       #"AV-40.28".FB_CLOSE := NOT #"AV-40.28".QCMD_OP;
       #"AV-40.29".FB_OPEN := #"AV-40.29".QCMD_OP;
       #"AV-40.29".FB_CLOSE := NOT #"AV-40.29".QCMD_OP;
       #"AV-40.30".FB_OPEN := #"AV-40.30".QCMD_OP;
       #"AV-40.30".FB_CLOSE := NOT #"AV-40.30".QCMD_OP;
       #"AV-40.31".FB_OPEN := #"AV-40.31".QCMD_OP;
       #"AV-40.31".FB_CLOSE := NOT #"AV-40.31".QCMD_OP;
       #"AV-40.32".FB_OPEN := #"AV-40.32".QCMD_OP;
       #"AV-40.32".FB_CLOSE := NOT #"AV-40.32".QCMD_OP;
       #"AV-40.33".FB_OPEN := #"AV-40.33".QCMD_OP;
       #"AV-40.33".FB_CLOSE := NOT #"AV-40.33".QCMD_OP;
       #"AV-40.34".FB_OPEN := #"AV-40.34".QCMD_OP;
       #"AV-40.34".FB_CLOSE := NOT #"AV-40.34".QCMD_OP;
   ELSE
       // Statement section ELSE
       #"AV-40.01".FB_OPEN := #"AV-40.01".QCMD_OP;
       #"AV-40.01".FB_CLOSE := NOT #"AV-40.01".QCMD_OP;
       #"AV-40.02".FB_OPEN := NOT "ZSC-40.02";
       #"AV-40.02".FB_CLOSE := "ZSC-40.02";
       #"AV-40.03".FB_OPEN := NOT "ZSC-40.03";
       #"AV-40.03".FB_CLOSE := "ZSC-40.03";
       #"AV-40.04".FB_OPEN := #"AV-40.04".QCMD_OP;
       #"AV-40.04".FB_CLOSE := NOT #"AV-40.04".QCMD_OP;
       #"AV-40.05".FB_OPEN := NOT "ZSC-40.05";
       #"AV-40.05".FB_CLOSE := "ZSC-40.05";
       #"AV-40.06".FB_OPEN := NOT "ZSC-40.06";
       #"AV-40.06".FB_CLOSE := "ZSC-40.06";
       #"AV-40.07".FB_OPEN := #"AV-40.07".QCMD_OP;
       #"AV-40.07".FB_CLOSE := NOT #"AV-40.07".QCMD_OP;
       #"AV-40.08".FB_OPEN := NOT "ZSC-40.08";
       #"AV-40.08".FB_CLOSE := "ZSC-40.08";
       #"AV-40.09".FB_OPEN := NOT "ZSC-40.09";
       #"AV-40.09".FB_CLOSE := "ZSC-40.09";
       #"AV-40.10".FB_OPEN := #"AV-40.10".QCMD_OP;
       #"AV-40.10".FB_CLOSE := NOT #"AV-40.10".QCMD_OP;
       #"AV-40.11".FB_OPEN := NOT "ZSC-40.11";
       #"AV-40.11".FB_CLOSE := "ZSC-40.11";
       #"AV-40.21".FB_OPEN := NOT "ZSC-40.21";
       #"AV-40.21".FB_CLOSE := "ZSC-40.21";
       #"AV-40.22".FB_OPEN := #"AV-40.22".QCMD_OP;
       #"AV-40.22".FB_CLOSE := NOT #"AV-40.22".QCMD_OP;
       #"AV-40.23".FB_OPEN := NOT "ZSC-40.23";
       #"AV-40.23".FB_CLOSE := "ZSC-40.23";
       #"AV-40.24".FB_OPEN := NOT "ZSC-40.24";
       #"AV-40.24".FB_CLOSE := "ZSC-40.24";
       #"AV-40.25".FB_OPEN := NOT "ZSC-40.25";
       #"AV-40.25".FB_CLOSE := "ZSC-40.25";
       #"AV-40.26".FB_OPEN := #"AV-40.26".QCMD_OP;
       #"AV-40.26".FB_CLOSE := NOT #"AV-40.26".QCMD_OP;
       #"AV-40.27".FB_OPEN := NOT "ZSC-40.27";
       #"AV-40.27".FB_CLOSE := "ZSC-40.27";
       #"AV-40.28".FB_OPEN := NOT "ZSC-40.28";
       #"AV-40.28".FB_CLOSE := "ZSC-40.28";
       #"AV-40.29".FB_OPEN := #"AV-40.29".QCMD_OP;
       #"AV-40.29".FB_CLOSE := NOT #"AV-40.29".QCMD_OP;
       #"AV-40.30".FB_OPEN := #"AV-40.30".QCMD_OP;
       #"AV-40.30".FB_CLOSE := NOT #"AV-40.30".QCMD_OP;
       #"AV-40.31".FB_OPEN := NOT "ZSC-40.31";
       #"AV-40.31".FB_CLOSE := "ZSC-40.31";
       #"AV-40.32".FB_OPEN := NOT "ZSC-40.32";
       #"AV-40.32".FB_CLOSE := "ZSC-40.32";
       #"AV-40.33".FB_OPEN := NOT "ZSC-40.33";
       #"AV-40.33".FB_CLOSE := "ZSC-40.33";
       #"AV-40.34".FB_OPEN := NOT "ZSC-40.34";
       #"AV-40.34".FB_CLOSE := "ZSC-40.34";
   END_IF;
END_REGION

NETWORK
TITLE = FB MONITORING TIME VALVE T-40
// FB OPEN TIME
      L     T#20s;
      T     #"AV-40.01".MON_T;
      T     #"AV-40.02".MON_T;
      T     #"AV-40.03".MON_T;
      T     #"AV-40.04".MON_T;
      T     #"AV-40.05".MON_T;
      T     #"AV-40.06".MON_T;
      T     #"AV-40.07".MON_T;
      T     #"AV-40.08".MON_T;
      T     #"AV-40.09".MON_T;
      T     #"AV-40.10".MON_T;
      T     #"AV-40.11".MON_T;
      T     #"AV-40.21".MON_T;
      T     #"AV-40.22".MON_T;
      T     #"AV-40.23".MON_T;
      T     #"AV-40.24".MON_T;
      T     #"AV-40.25".MON_T;
      T     #"AV-40.26".MON_T;
      T     #"AV-40.27".MON_T;
      T     #"AV-40.28".MON_T;
      T     #"AV-40.29".MON_T;
      T     #"AV-40.30".MON_T;
      T     #"AV-40.31".MON_T;
      T     #"AV-40.32".MON_T;
      T     #"AV-40.33".MON_T;
      T     #"AV-40.34".MON_T;

// FB CLOSE TIME
      L     T#20s;
      T     #"AV-40.01".MON_T_CLOSE;
      T     #"AV-40.02".MON_T_CLOSE;
      T     #"AV-40.03".MON_T_CLOSE;
      T     #"AV-40.04".MON_T_CLOSE;
      T     #"AV-40.05".MON_T_CLOSE;
      T     #"AV-40.06".MON_T_CLOSE;
      T     #"AV-40.07".MON_T_CLOSE;
      T     #"AV-40.08".MON_T_CLOSE;
      T     #"AV-40.09".MON_T_CLOSE;
      T     #"AV-40.10".MON_T_CLOSE;
      T     #"AV-40.11".MON_T_CLOSE;
      T     #"AV-40.21".MON_T_CLOSE;
      T     #"AV-40.22".MON_T_CLOSE;
      T     #"AV-40.23".MON_T_CLOSE;
      T     #"AV-40.24".MON_T_CLOSE;
      T     #"AV-40.25".MON_T_CLOSE;
      T     #"AV-40.26".MON_T_CLOSE;
      T     #"AV-40.27".MON_T_CLOSE;
      T     #"AV-40.28".MON_T_CLOSE;
      T     #"AV-40.29".MON_T_CLOSE;
      T     #"AV-40.30".MON_T_CLOSE;
      T     #"AV-40.31".MON_T_CLOSE;
      T     #"AV-40.32".MON_T_CLOSE;
      T     #"AV-40.33".MON_T_CLOSE;
      T     #"AV-40.34".MON_T_CLOSE;


REGION Network 4: AV-40.01
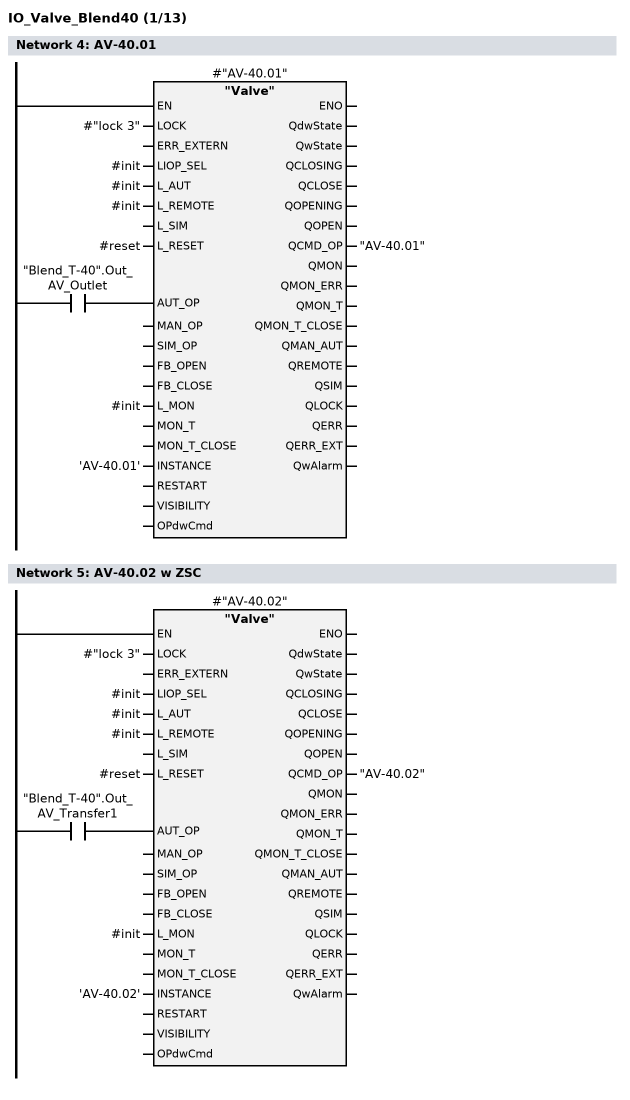
   RUNG wire#powerrail
      #"AV-40.01"(AUT_OP := wire#w1, LOCK := #"lock 3", ERR_EXTERN :=, LIOP_SEL := #init, L_AUT := #init, L_REMOTE := #init, L_SIM :=, L_RESET := #reset, MAN_OP :=, SIM_OP :=, FB_OPEN :=, FB_CLOSE :=, L_MON := #init, MON_T :=, MON_T_CLOSE :=, INSTANCE := 'AV-40.01', RESTART :=, VISIBILITY :=, OPdwCmd :=, QdwState =>, QwState =>, QCLOSING =>, QCLOSE =>, QOPENING =>, QOPEN =>, QCMD_OP => "AV-40.01", QMON =>, QMON_ERR =>, QMON_T =>, QMON_T_CLOSE =>, QMAN_AUT =>, QREMOTE =>, QSIM =>, QLOCK =>, QERR =>, QERR_EXT =>, QwAlarm =>)
   END_RUNG
   RUNG wire#powerrail
      Contact( "Blend_T-40".Out_AV_Outlet )
   END_RUNG wire#w1
   // the same network as SCL:
   #"AV-40.01"(LOCK := #"lock 3",   // "Valve"
               LIOP_SEL := #init,
               L_AUT := #init,
               L_REMOTE := #init,
               L_RESET := #reset,
               AUT_OP := "Blend_T-40".Out_AV_Outlet,
               L_MON := #init,
               INSTANCE := 'AV-40.01',
               QCMD_OP => "AV-40.01");
END_REGION

REGION Network 5: AV-40.02 w ZSC
   RUNG wire#powerrail
      #"AV-40.02"(AUT_OP := wire#w1, LOCK := #"lock 3", ERR_EXTERN :=, LIOP_SEL := #init, L_AUT := #init, L_REMOTE := #init, L_SIM :=, L_RESET := #reset, MAN_OP :=, SIM_OP :=, FB_OPEN :=, FB_CLOSE :=, L_MON := #init, MON_T :=, MON_T_CLOSE :=, INSTANCE := 'AV-40.02', RESTART :=, VISIBILITY :=, OPdwCmd :=, QdwState =>, QwState =>, QCLOSING =>, QCLOSE =>, QOPENING =>, QOPEN =>, QCMD_OP => "AV-40.02", QMON =>, QMON_ERR =>, QMON_T =>, QMON_T_CLOSE =>, QMAN_AUT =>, QREMOTE =>, QSIM =>, QLOCK =>, QERR =>, QERR_EXT =>, QwAlarm =>)
   END_RUNG
   RUNG wire#powerrail
      Contact( "Blend_T-40".Out_AV_Transfer1 )
   END_RUNG wire#w1
   // the same network as SCL:
   #"AV-40.02"(LOCK := #"lock 3",   // "Valve"
               LIOP_SEL := #init,
               L_AUT := #init,
               L_REMOTE := #init,
               L_RESET := #reset,
               AUT_OP := "Blend_T-40".Out_AV_Transfer1,
               L_MON := #init,
               INSTANCE := 'AV-40.02',
               QCMD_OP => "AV-40.02");
END_REGION

REGION Network 6: AV-40.03 w ZSC
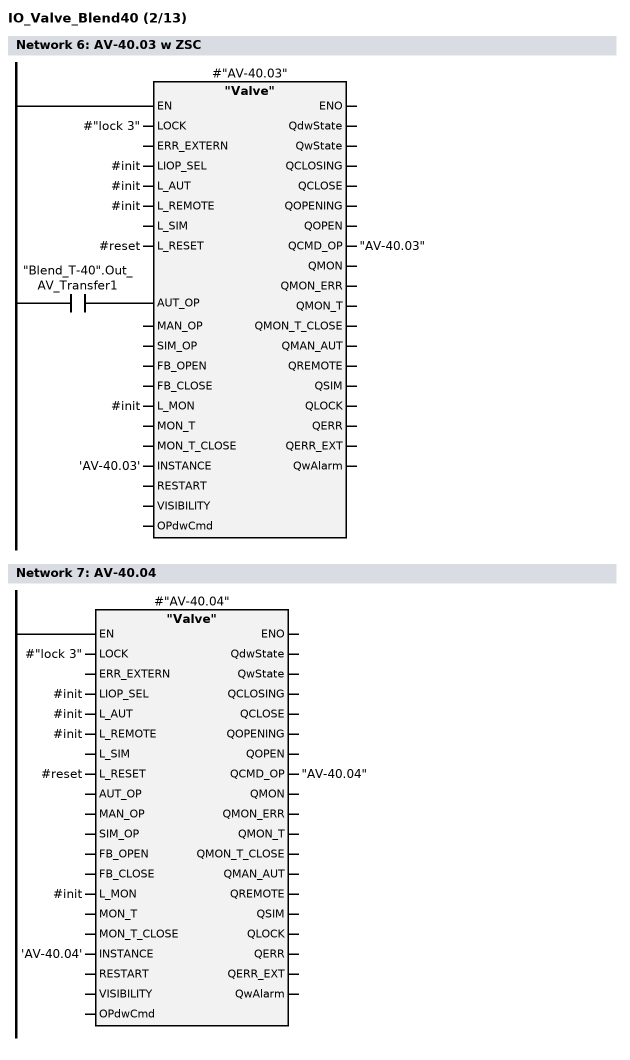
   RUNG wire#powerrail
      #"AV-40.03"(AUT_OP := wire#w1, LOCK := #"lock 3", ERR_EXTERN :=, LIOP_SEL := #init, L_AUT := #init, L_REMOTE := #init, L_SIM :=, L_RESET := #reset, MAN_OP :=, SIM_OP :=, FB_OPEN :=, FB_CLOSE :=, L_MON := #init, MON_T :=, MON_T_CLOSE :=, INSTANCE := 'AV-40.03', RESTART :=, VISIBILITY :=, OPdwCmd :=, QdwState =>, QwState =>, QCLOSING =>, QCLOSE =>, QOPENING =>, QOPEN =>, QCMD_OP => "AV-40.03", QMON =>, QMON_ERR =>, QMON_T =>, QMON_T_CLOSE =>, QMAN_AUT =>, QREMOTE =>, QSIM =>, QLOCK =>, QERR =>, QERR_EXT =>, QwAlarm =>)
   END_RUNG
   RUNG wire#powerrail
      Contact( "Blend_T-40".Out_AV_Transfer1 )
   END_RUNG wire#w1
   // the same network as SCL:
   #"AV-40.03"(LOCK := #"lock 3",   // "Valve"
               LIOP_SEL := #init,
               L_AUT := #init,
               L_REMOTE := #init,
               L_RESET := #reset,
               AUT_OP := "Blend_T-40".Out_AV_Transfer1,
               L_MON := #init,
               INSTANCE := 'AV-40.03',
               QCMD_OP => "AV-40.03");
END_REGION

REGION Network 7: AV-40.04
   RUNG wire#powerrail
      #"AV-40.04"(LOCK := #"lock 3", ERR_EXTERN :=, LIOP_SEL := #init, L_AUT := #init, L_REMOTE := #init, L_SIM :=, L_RESET := #reset, AUT_OP :=, MAN_OP :=, SIM_OP :=, FB_OPEN :=, FB_CLOSE :=, L_MON := #init, MON_T :=, MON_T_CLOSE :=, INSTANCE := 'AV-40.04', RESTART :=, VISIBILITY :=, OPdwCmd :=, QdwState =>, QwState =>, QCLOSING =>, QCLOSE =>, QOPENING =>, QOPEN =>, QCMD_OP => "AV-40.04", QMON =>, QMON_ERR =>, QMON_T =>, QMON_T_CLOSE =>, QMAN_AUT =>, QREMOTE =>, QSIM =>, QLOCK =>, QERR =>, QERR_EXT =>, QwAlarm =>)
   END_RUNG
   // the same network as SCL:
   #"AV-40.04"(LOCK := #"lock 3",   // "Valve"
               LIOP_SEL := #init,
               L_AUT := #init,
               L_REMOTE := #init,
               L_RESET := #reset,
               L_MON := #init,
               INSTANCE := 'AV-40.04',
               QCMD_OP => "AV-40.04");
END_REGION

REGION Network 8: AV-40.05 w ZSC
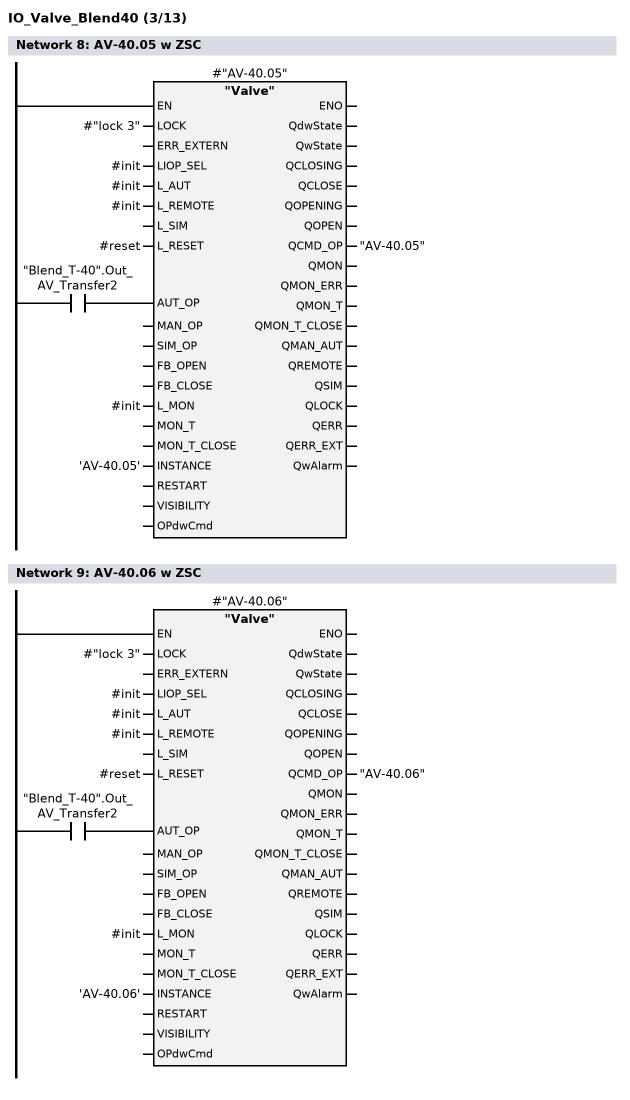
   RUNG wire#powerrail
      #"AV-40.05"(AUT_OP := wire#w1, LOCK := #"lock 3", ERR_EXTERN :=, LIOP_SEL := #init, L_AUT := #init, L_REMOTE := #init, L_SIM :=, L_RESET := #reset, MAN_OP :=, SIM_OP :=, FB_OPEN :=, FB_CLOSE :=, L_MON := #init, MON_T :=, MON_T_CLOSE :=, INSTANCE := 'AV-40.05', RESTART :=, VISIBILITY :=, OPdwCmd :=, QdwState =>, QwState =>, QCLOSING =>, QCLOSE =>, QOPENING =>, QOPEN =>, QCMD_OP => "AV-40.05", QMON =>, QMON_ERR =>, QMON_T =>, QMON_T_CLOSE =>, QMAN_AUT =>, QREMOTE =>, QSIM =>, QLOCK =>, QERR =>, QERR_EXT =>, QwAlarm =>)
   END_RUNG
   RUNG wire#powerrail
      Contact( "Blend_T-40".Out_AV_Transfer2 )
   END_RUNG wire#w1
   // the same network as SCL:
   #"AV-40.05"(LOCK := #"lock 3",   // "Valve"
               LIOP_SEL := #init,
               L_AUT := #init,
               L_REMOTE := #init,
               L_RESET := #reset,
               AUT_OP := "Blend_T-40".Out_AV_Transfer2,
               L_MON := #init,
               INSTANCE := 'AV-40.05',
               QCMD_OP => "AV-40.05");
END_REGION

REGION Network 9: AV-40.06 w ZSC
   RUNG wire#powerrail
      #"AV-40.06"(AUT_OP := wire#w1, LOCK := #"lock 3", ERR_EXTERN :=, LIOP_SEL := #init, L_AUT := #init, L_REMOTE := #init, L_SIM :=, L_RESET := #reset, MAN_OP :=, SIM_OP :=, FB_OPEN :=, FB_CLOSE :=, L_MON := #init, MON_T :=, MON_T_CLOSE :=, INSTANCE := 'AV-40.06', RESTART :=, VISIBILITY :=, OPdwCmd :=, QdwState =>, QwState =>, QCLOSING =>, QCLOSE =>, QOPENING =>, QOPEN =>, QCMD_OP => "AV-40.06", QMON =>, QMON_ERR =>, QMON_T =>, QMON_T_CLOSE =>, QMAN_AUT =>, QREMOTE =>, QSIM =>, QLOCK =>, QERR =>, QERR_EXT =>, QwAlarm =>)
   END_RUNG
   RUNG wire#powerrail
      Contact( "Blend_T-40".Out_AV_Transfer2 )
   END_RUNG wire#w1
   // the same network as SCL:
   #"AV-40.06"(LOCK := #"lock 3",   // "Valve"
               LIOP_SEL := #init,
               L_AUT := #init,
               L_REMOTE := #init,
               L_RESET := #reset,
               AUT_OP := "Blend_T-40".Out_AV_Transfer2,
               L_MON := #init,
               INSTANCE := 'AV-40.06',
               QCMD_OP => "AV-40.06");
END_REGION

REGION Network 10: AV-40.07
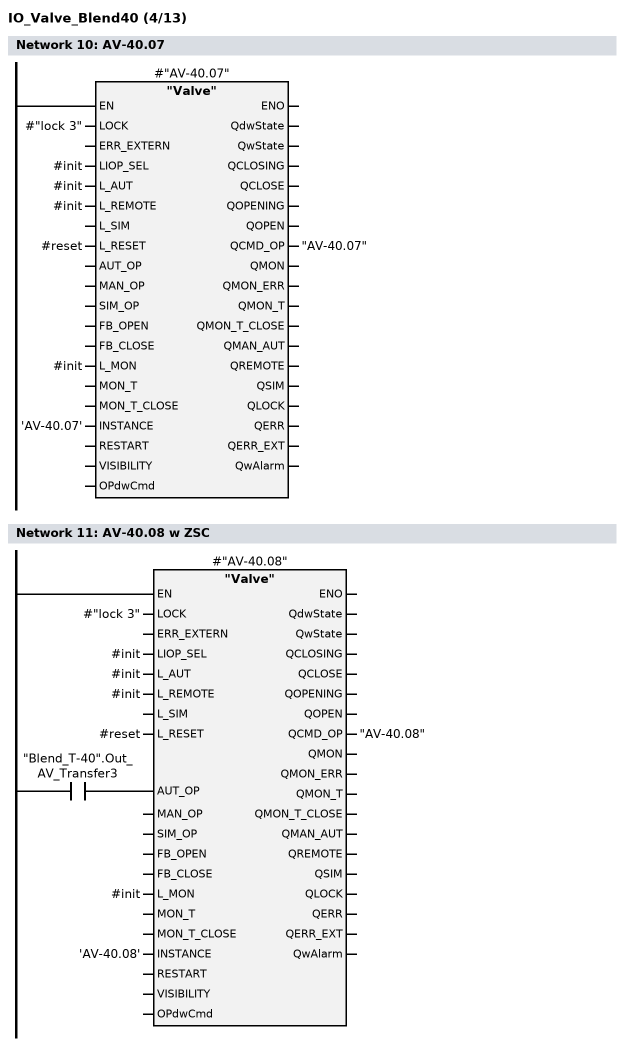
   RUNG wire#powerrail
      #"AV-40.07"(LOCK := #"lock 3", ERR_EXTERN :=, LIOP_SEL := #init, L_AUT := #init, L_REMOTE := #init, L_SIM :=, L_RESET := #reset, AUT_OP :=, MAN_OP :=, SIM_OP :=, FB_OPEN :=, FB_CLOSE :=, L_MON := #init, MON_T :=, MON_T_CLOSE :=, INSTANCE := 'AV-40.07', RESTART :=, VISIBILITY :=, OPdwCmd :=, QdwState =>, QwState =>, QCLOSING =>, QCLOSE =>, QOPENING =>, QOPEN =>, QCMD_OP => "AV-40.07", QMON =>, QMON_ERR =>, QMON_T =>, QMON_T_CLOSE =>, QMAN_AUT =>, QREMOTE =>, QSIM =>, QLOCK =>, QERR =>, QERR_EXT =>, QwAlarm =>)
   END_RUNG
   // the same network as SCL:
   #"AV-40.07"(LOCK := #"lock 3",   // "Valve"
               LIOP_SEL := #init,
               L_AUT := #init,
               L_REMOTE := #init,
               L_RESET := #reset,
               L_MON := #init,
               INSTANCE := 'AV-40.07',
               QCMD_OP => "AV-40.07");
END_REGION

REGION Network 11: AV-40.08 w ZSC
   RUNG wire#powerrail
      #"AV-40.08"(AUT_OP := wire#w1, LOCK := #"lock 3", ERR_EXTERN :=, LIOP_SEL := #init, L_AUT := #init, L_REMOTE := #init, L_SIM :=, L_RESET := #reset, MAN_OP :=, SIM_OP :=, FB_OPEN :=, FB_CLOSE :=, L_MON := #init, MON_T :=, MON_T_CLOSE :=, INSTANCE := 'AV-40.08', RESTART :=, VISIBILITY :=, OPdwCmd :=, QdwState =>, QwState =>, QCLOSING =>, QCLOSE =>, QOPENING =>, QOPEN =>, QCMD_OP => "AV-40.08", QMON =>, QMON_ERR =>, QMON_T =>, QMON_T_CLOSE =>, QMAN_AUT =>, QREMOTE =>, QSIM =>, QLOCK =>, QERR =>, QERR_EXT =>, QwAlarm =>)
   END_RUNG
   RUNG wire#powerrail
      Contact( "Blend_T-40".Out_AV_Transfer3 )
   END_RUNG wire#w1
   // the same network as SCL:
   #"AV-40.08"(LOCK := #"lock 3",   // "Valve"
               LIOP_SEL := #init,
               L_AUT := #init,
               L_REMOTE := #init,
               L_RESET := #reset,
               AUT_OP := "Blend_T-40".Out_AV_Transfer3,
               L_MON := #init,
               INSTANCE := 'AV-40.08',
               QCMD_OP => "AV-40.08");
END_REGION

REGION Network 12: AV-40.09 w ZSC
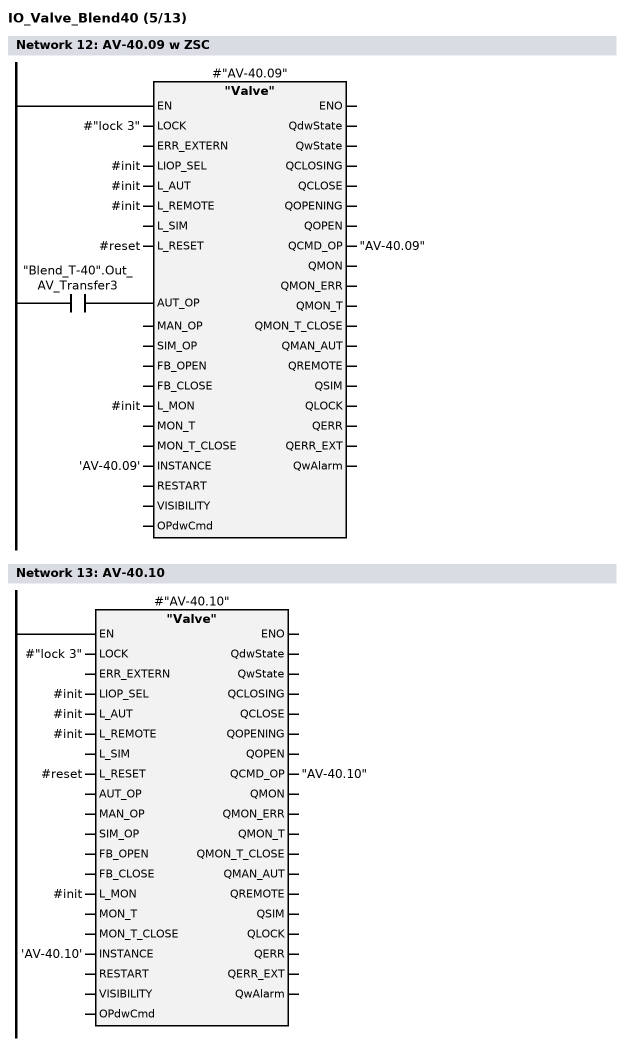
   RUNG wire#powerrail
      #"AV-40.09"(AUT_OP := wire#w1, LOCK := #"lock 3", ERR_EXTERN :=, LIOP_SEL := #init, L_AUT := #init, L_REMOTE := #init, L_SIM :=, L_RESET := #reset, MAN_OP :=, SIM_OP :=, FB_OPEN :=, FB_CLOSE :=, L_MON := #init, MON_T :=, MON_T_CLOSE :=, INSTANCE := 'AV-40.09', RESTART :=, VISIBILITY :=, OPdwCmd :=, QdwState =>, QwState =>, QCLOSING =>, QCLOSE =>, QOPENING =>, QOPEN =>, QCMD_OP => "AV-40.09", QMON =>, QMON_ERR =>, QMON_T =>, QMON_T_CLOSE =>, QMAN_AUT =>, QREMOTE =>, QSIM =>, QLOCK =>, QERR =>, QERR_EXT =>, QwAlarm =>)
   END_RUNG
   RUNG wire#powerrail
      Contact( "Blend_T-40".Out_AV_Transfer3 )
   END_RUNG wire#w1
   // the same network as SCL:
   #"AV-40.09"(LOCK := #"lock 3",   // "Valve"
               LIOP_SEL := #init,
               L_AUT := #init,
               L_REMOTE := #init,
               L_RESET := #reset,
               AUT_OP := "Blend_T-40".Out_AV_Transfer3,
               L_MON := #init,
               INSTANCE := 'AV-40.09',
               QCMD_OP => "AV-40.09");
END_REGION

REGION Network 13: AV-40.10
   RUNG wire#powerrail
      #"AV-40.10"(LOCK := #"lock 3", ERR_EXTERN :=, LIOP_SEL := #init, L_AUT := #init, L_REMOTE := #init, L_SIM :=, L_RESET := #reset, AUT_OP :=, MAN_OP :=, SIM_OP :=, FB_OPEN :=, FB_CLOSE :=, L_MON := #init, MON_T :=, MON_T_CLOSE :=, INSTANCE := 'AV-40.10', RESTART :=, VISIBILITY :=, OPdwCmd :=, QdwState =>, QwState =>, QCLOSING =>, QCLOSE =>, QOPENING =>, QOPEN =>, QCMD_OP => "AV-40.10", QMON =>, QMON_ERR =>, QMON_T =>, QMON_T_CLOSE =>, QMAN_AUT =>, QREMOTE =>, QSIM =>, QLOCK =>, QERR =>, QERR_EXT =>, QwAlarm =>)
   END_RUNG
   // the same network as SCL:
   #"AV-40.10"(LOCK := #"lock 3",   // "Valve"
               LIOP_SEL := #init,
               L_AUT := #init,
               L_REMOTE := #init,
               L_RESET := #reset,
               L_MON := #init,
               INSTANCE := 'AV-40.10',
               QCMD_OP => "AV-40.10");
END_REGION

REGION Network 14: AV-40.11 w ZSC
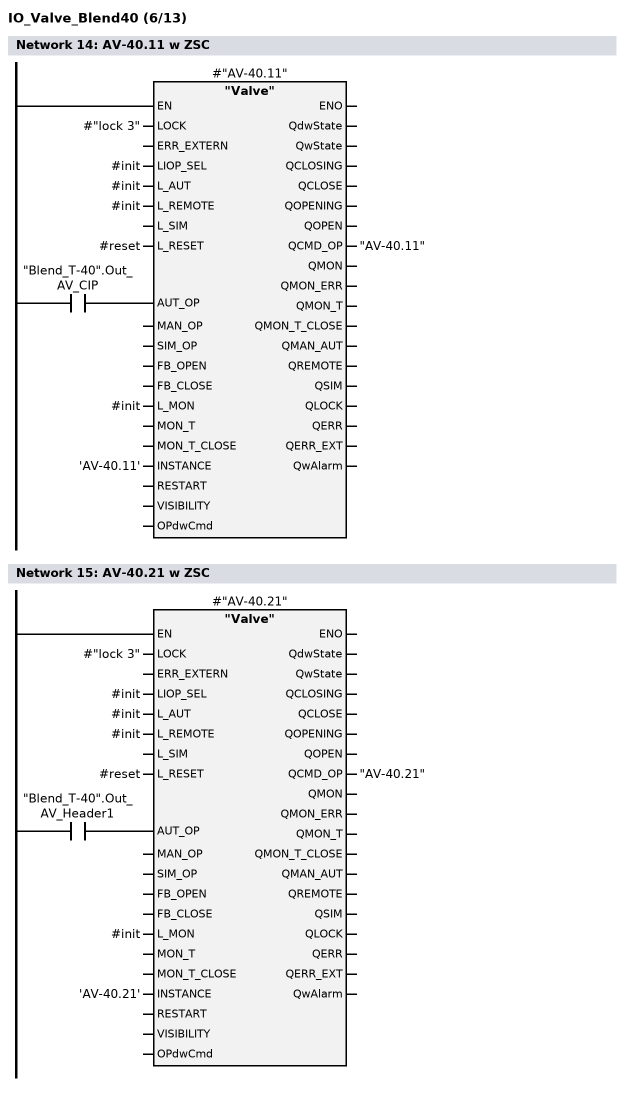
   RUNG wire#powerrail
      #"AV-40.11"(AUT_OP := wire#w1, LOCK := #"lock 3", ERR_EXTERN :=, LIOP_SEL := #init, L_AUT := #init, L_REMOTE := #init, L_SIM :=, L_RESET := #reset, MAN_OP :=, SIM_OP :=, FB_OPEN :=, FB_CLOSE :=, L_MON := #init, MON_T :=, MON_T_CLOSE :=, INSTANCE := 'AV-40.11', RESTART :=, VISIBILITY :=, OPdwCmd :=, QdwState =>, QwState =>, QCLOSING =>, QCLOSE =>, QOPENING =>, QOPEN =>, QCMD_OP => "AV-40.11", QMON =>, QMON_ERR =>, QMON_T =>, QMON_T_CLOSE =>, QMAN_AUT =>, QREMOTE =>, QSIM =>, QLOCK =>, QERR =>, QERR_EXT =>, QwAlarm =>)
   END_RUNG
   RUNG wire#powerrail
      Contact( "Blend_T-40".Out_AV_CIP )
   END_RUNG wire#w1
   // the same network as SCL:
   #"AV-40.11"(LOCK := #"lock 3",   // "Valve"
               LIOP_SEL := #init,
               L_AUT := #init,
               L_REMOTE := #init,
               L_RESET := #reset,
               AUT_OP := "Blend_T-40".Out_AV_CIP,
               L_MON := #init,
               INSTANCE := 'AV-40.11',
               QCMD_OP => "AV-40.11");
END_REGION

REGION Network 15: AV-40.21 w ZSC
   RUNG wire#powerrail
      #"AV-40.21"(AUT_OP := wire#w1, LOCK := #"lock 3", ERR_EXTERN :=, LIOP_SEL := #init, L_AUT := #init, L_REMOTE := #init, L_SIM :=, L_RESET := #reset, MAN_OP :=, SIM_OP :=, FB_OPEN :=, FB_CLOSE :=, L_MON := #init, MON_T :=, MON_T_CLOSE :=, INSTANCE := 'AV-40.21', RESTART :=, VISIBILITY :=, OPdwCmd :=, QdwState =>, QwState =>, QCLOSING =>, QCLOSE =>, QOPENING =>, QOPEN =>, QCMD_OP => "AV-40.21", QMON =>, QMON_ERR =>, QMON_T =>, QMON_T_CLOSE =>, QMAN_AUT =>, QREMOTE =>, QSIM =>, QLOCK =>, QERR =>, QERR_EXT =>, QwAlarm =>)
   END_RUNG
   RUNG wire#powerrail
      Contact( "Blend_T-40".Out_AV_Header1 )
   END_RUNG wire#w1
   // the same network as SCL:
   #"AV-40.21"(LOCK := #"lock 3",   // "Valve"
               LIOP_SEL := #init,
               L_AUT := #init,
               L_REMOTE := #init,
               L_RESET := #reset,
               AUT_OP := "Blend_T-40".Out_AV_Header1,
               L_MON := #init,
               INSTANCE := 'AV-40.21',
               QCMD_OP => "AV-40.21");
END_REGION

REGION Network 16: AV-40.22
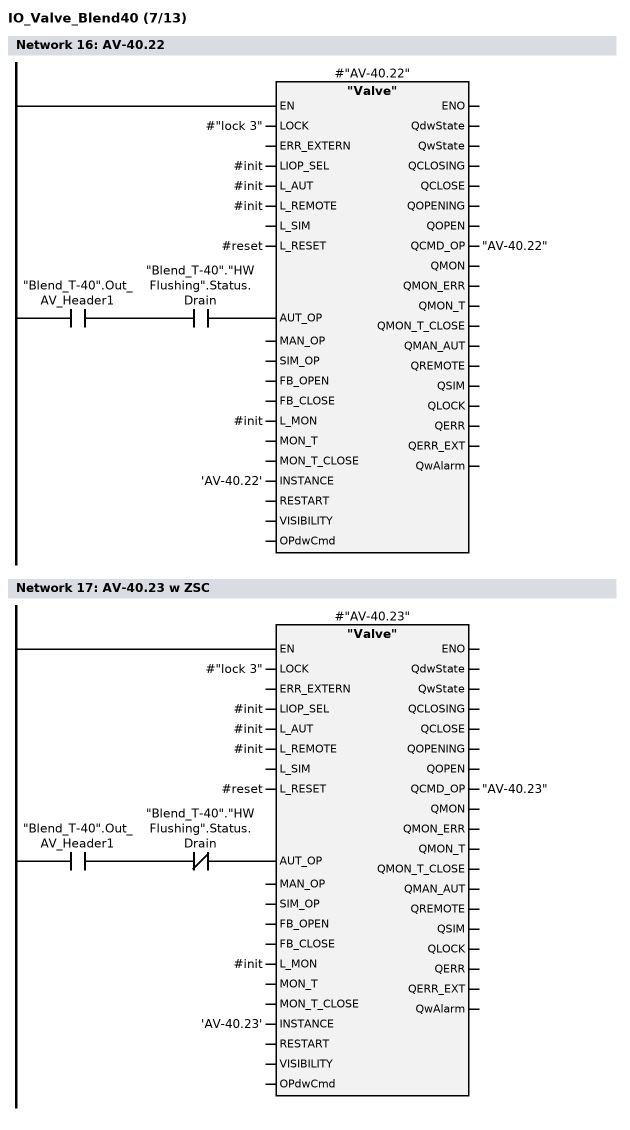
   RUNG wire#powerrail
      #"AV-40.22"(AUT_OP := wire#w1, LOCK := #"lock 3", ERR_EXTERN :=, LIOP_SEL := #init, L_AUT := #init, L_REMOTE := #init, L_SIM :=, L_RESET := #reset, MAN_OP :=, SIM_OP :=, FB_OPEN :=, FB_CLOSE :=, L_MON := #init, MON_T :=, MON_T_CLOSE :=, INSTANCE := 'AV-40.22', RESTART :=, VISIBILITY :=, OPdwCmd :=, QdwState =>, QwState =>, QCLOSING =>, QCLOSE =>, QOPENING =>, QOPEN =>, QCMD_OP => "AV-40.22", QMON =>, QMON_ERR =>, QMON_T =>, QMON_T_CLOSE =>, QMAN_AUT =>, QREMOTE =>, QSIM =>, QLOCK =>, QERR =>, QERR_EXT =>, QwAlarm =>)
   END_RUNG
   RUNG wire#powerrail
      Contact( "Blend_T-40".Out_AV_Header1 )
      Contact( "Blend_T-40"."HW Flushing".Status.Drain )
   END_RUNG wire#w1
   // the same network as SCL:
   #"AV-40.22"(LOCK := #"lock 3",   // "Valve"
               LIOP_SEL := #init,
               L_AUT := #init,
               L_REMOTE := #init,
               L_RESET := #reset,
               AUT_OP := "Blend_T-40".Out_AV_Header1 AND "Blend_T-40"."HW Flushing".Status.Drain,
               L_MON := #init,
               INSTANCE := 'AV-40.22',
               QCMD_OP => "AV-40.22");
END_REGION

REGION Network 17: AV-40.23 w ZSC
   RUNG wire#powerrail
      #"AV-40.23"(AUT_OP := wire#w1, LOCK := #"lock 3", ERR_EXTERN :=, LIOP_SEL := #init, L_AUT := #init, L_REMOTE := #init, L_SIM :=, L_RESET := #reset, MAN_OP :=, SIM_OP :=, FB_OPEN :=, FB_CLOSE :=, L_MON := #init, MON_T :=, MON_T_CLOSE :=, INSTANCE := 'AV-40.23', RESTART :=, VISIBILITY :=, OPdwCmd :=, QdwState =>, QwState =>, QCLOSING =>, QCLOSE =>, QOPENING =>, QOPEN =>, QCMD_OP => "AV-40.23", QMON =>, QMON_ERR =>, QMON_T =>, QMON_T_CLOSE =>, QMAN_AUT =>, QREMOTE =>, QSIM =>, QLOCK =>, QERR =>, QERR_EXT =>, QwAlarm =>)
   END_RUNG
   RUNG wire#powerrail
      Contact( "Blend_T-40".Out_AV_Header1 )
      I_Contact( "Blend_T-40"."HW Flushing".Status.Drain )
   END_RUNG wire#w1
   // the same network as SCL:
   #"AV-40.23"(LOCK := #"lock 3",   // "Valve"
               LIOP_SEL := #init,
               L_AUT := #init,
               L_REMOTE := #init,
               L_RESET := #reset,
               AUT_OP := "Blend_T-40".Out_AV_Header1 AND NOT "Blend_T-40"."HW Flushing".Status.Drain,
               L_MON := #init,
               INSTANCE := 'AV-40.23',
               QCMD_OP => "AV-40.23");
END_REGION

REGION Network 18: AV-40.24 w ZSC
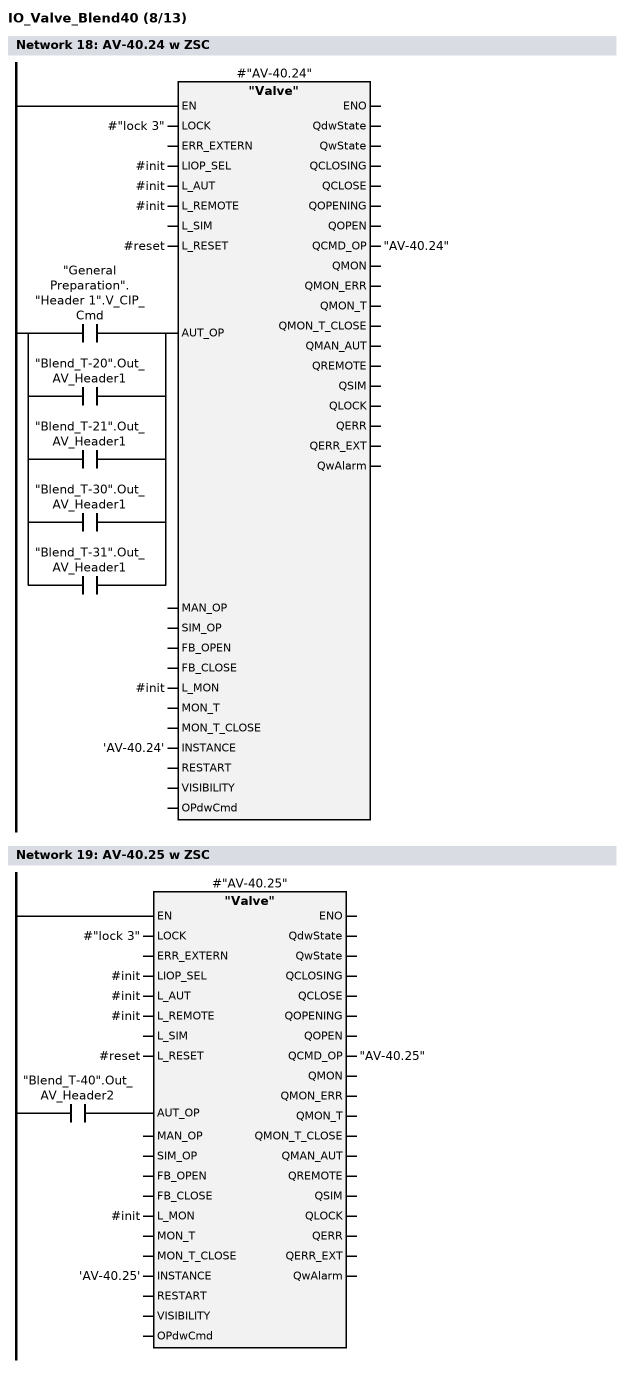
   RUNG wire#powerrail
      #"AV-40.24"(AUT_OP := wire#w1, LOCK := #"lock 3", ERR_EXTERN :=, LIOP_SEL := #init, L_AUT := #init, L_REMOTE := #init, L_SIM :=, L_RESET := #reset, MAN_OP :=, SIM_OP :=, FB_OPEN :=, FB_CLOSE :=, L_MON := #init, MON_T :=, MON_T_CLOSE :=, INSTANCE := 'AV-40.24', RESTART :=, VISIBILITY :=, OPdwCmd :=, QdwState =>, QwState =>, QCLOSING =>, QCLOSE =>, QOPENING =>, QOPEN =>, QCMD_OP => "AV-40.24", QMON =>, QMON_ERR =>, QMON_T =>, QMON_T_CLOSE =>, QMAN_AUT =>, QREMOTE =>, QSIM =>, QLOCK =>, QERR =>, QERR_EXT =>, QwAlarm =>)
   END_RUNG
   RUNG wire#powerrail
      Contact( "General Preparation"."Header 1".V_CIP_Cmd )
   END_RUNG wire#w1
   RUNG wire#powerrail
      Contact( "Blend_T-20".Out_AV_Header1 )
   END_RUNG wire#w1
   RUNG wire#powerrail
      Contact( "Blend_T-21".Out_AV_Header1 )
   END_RUNG wire#w1
   RUNG wire#powerrail
      Contact( "Blend_T-30".Out_AV_Header1 )
   END_RUNG wire#w1
   RUNG wire#powerrail
      Contact( "Blend_T-31".Out_AV_Header1 )
   END_RUNG wire#w1
   // the same network as SCL:
   #"AV-40.24"(LOCK := #"lock 3",   // "Valve"
               LIOP_SEL := #init,
               L_AUT := #init,
               L_REMOTE := #init,
               L_RESET := #reset,
               AUT_OP := "General Preparation"."Header 1".V_CIP_Cmd OR "Blend_T-20".Out_AV_Header1 OR "Blend_T-21".Out_AV_Header1 OR "Blend_T-30".Out_AV_Header1 OR "Blend_T-31".Out_AV_Header1,
               L_MON := #init,
               INSTANCE := 'AV-40.24',
               QCMD_OP => "AV-40.24");
END_REGION

REGION Network 19: AV-40.25 w ZSC
   RUNG wire#powerrail
      #"AV-40.25"(AUT_OP := wire#w1, LOCK := #"lock 3", ERR_EXTERN :=, LIOP_SEL := #init, L_AUT := #init, L_REMOTE := #init, L_SIM :=, L_RESET := #reset, MAN_OP :=, SIM_OP :=, FB_OPEN :=, FB_CLOSE :=, L_MON := #init, MON_T :=, MON_T_CLOSE :=, INSTANCE := 'AV-40.25', RESTART :=, VISIBILITY :=, OPdwCmd :=, QdwState =>, QwState =>, QCLOSING =>, QCLOSE =>, QOPENING =>, QOPEN =>, QCMD_OP => "AV-40.25", QMON =>, QMON_ERR =>, QMON_T =>, QMON_T_CLOSE =>, QMAN_AUT =>, QREMOTE =>, QSIM =>, QLOCK =>, QERR =>, QERR_EXT =>, QwAlarm =>)
   END_RUNG
   RUNG wire#powerrail
      Contact( "Blend_T-40".Out_AV_Header2 )
   END_RUNG wire#w1
   // the same network as SCL:
   #"AV-40.25"(LOCK := #"lock 3",   // "Valve"
               LIOP_SEL := #init,
               L_AUT := #init,
               L_REMOTE := #init,
               L_RESET := #reset,
               AUT_OP := "Blend_T-40".Out_AV_Header2,
               L_MON := #init,
               INSTANCE := 'AV-40.25',
               QCMD_OP => "AV-40.25");
END_REGION

REGION Network 20: AV-40.26
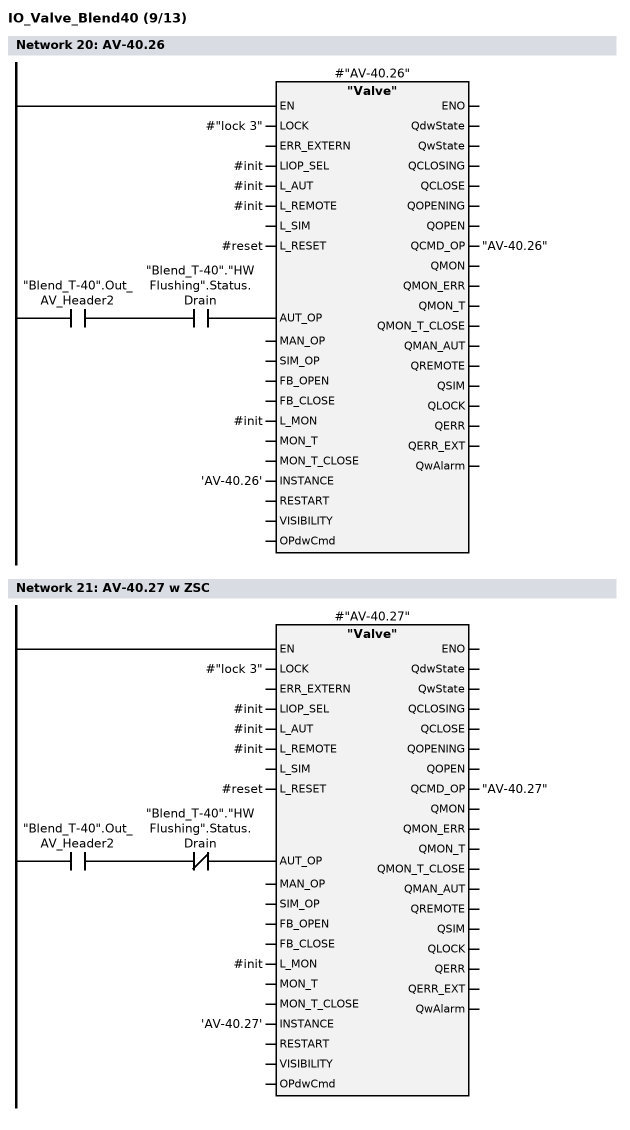
   RUNG wire#powerrail
      #"AV-40.26"(AUT_OP := wire#w1, LOCK := #"lock 3", ERR_EXTERN :=, LIOP_SEL := #init, L_AUT := #init, L_REMOTE := #init, L_SIM :=, L_RESET := #reset, MAN_OP :=, SIM_OP :=, FB_OPEN :=, FB_CLOSE :=, L_MON := #init, MON_T :=, MON_T_CLOSE :=, INSTANCE := 'AV-40.26', RESTART :=, VISIBILITY :=, OPdwCmd :=, QdwState =>, QwState =>, QCLOSING =>, QCLOSE =>, QOPENING =>, QOPEN =>, QCMD_OP => "AV-40.26", QMON =>, QMON_ERR =>, QMON_T =>, QMON_T_CLOSE =>, QMAN_AUT =>, QREMOTE =>, QSIM =>, QLOCK =>, QERR =>, QERR_EXT =>, QwAlarm =>)
   END_RUNG
   RUNG wire#powerrail
      Contact( "Blend_T-40".Out_AV_Header2 )
      Contact( "Blend_T-40"."HW Flushing".Status.Drain )
   END_RUNG wire#w1
   // the same network as SCL:
   #"AV-40.26"(LOCK := #"lock 3",   // "Valve"
               LIOP_SEL := #init,
               L_AUT := #init,
               L_REMOTE := #init,
               L_RESET := #reset,
               AUT_OP := "Blend_T-40".Out_AV_Header2 AND "Blend_T-40"."HW Flushing".Status.Drain,
               L_MON := #init,
               INSTANCE := 'AV-40.26',
               QCMD_OP => "AV-40.26");
END_REGION

REGION Network 21: AV-40.27 w ZSC
   RUNG wire#powerrail
      #"AV-40.27"(AUT_OP := wire#w1, LOCK := #"lock 3", ERR_EXTERN :=, LIOP_SEL := #init, L_AUT := #init, L_REMOTE := #init, L_SIM :=, L_RESET := #reset, MAN_OP :=, SIM_OP :=, FB_OPEN :=, FB_CLOSE :=, L_MON := #init, MON_T :=, MON_T_CLOSE :=, INSTANCE := 'AV-40.27', RESTART :=, VISIBILITY :=, OPdwCmd :=, QdwState =>, QwState =>, QCLOSING =>, QCLOSE =>, QOPENING =>, QOPEN =>, QCMD_OP => "AV-40.27", QMON =>, QMON_ERR =>, QMON_T =>, QMON_T_CLOSE =>, QMAN_AUT =>, QREMOTE =>, QSIM =>, QLOCK =>, QERR =>, QERR_EXT =>, QwAlarm =>)
   END_RUNG
   RUNG wire#powerrail
      Contact( "Blend_T-40".Out_AV_Header2 )
      I_Contact( "Blend_T-40"."HW Flushing".Status.Drain )
   END_RUNG wire#w1
   // the same network as SCL:
   #"AV-40.27"(LOCK := #"lock 3",   // "Valve"
               LIOP_SEL := #init,
               L_AUT := #init,
               L_REMOTE := #init,
               L_RESET := #reset,
               AUT_OP := "Blend_T-40".Out_AV_Header2 AND NOT "Blend_T-40"."HW Flushing".Status.Drain,
               L_MON := #init,
               INSTANCE := 'AV-40.27',
               QCMD_OP => "AV-40.27");
END_REGION

REGION Network 22: AV-40.28 w ZSC
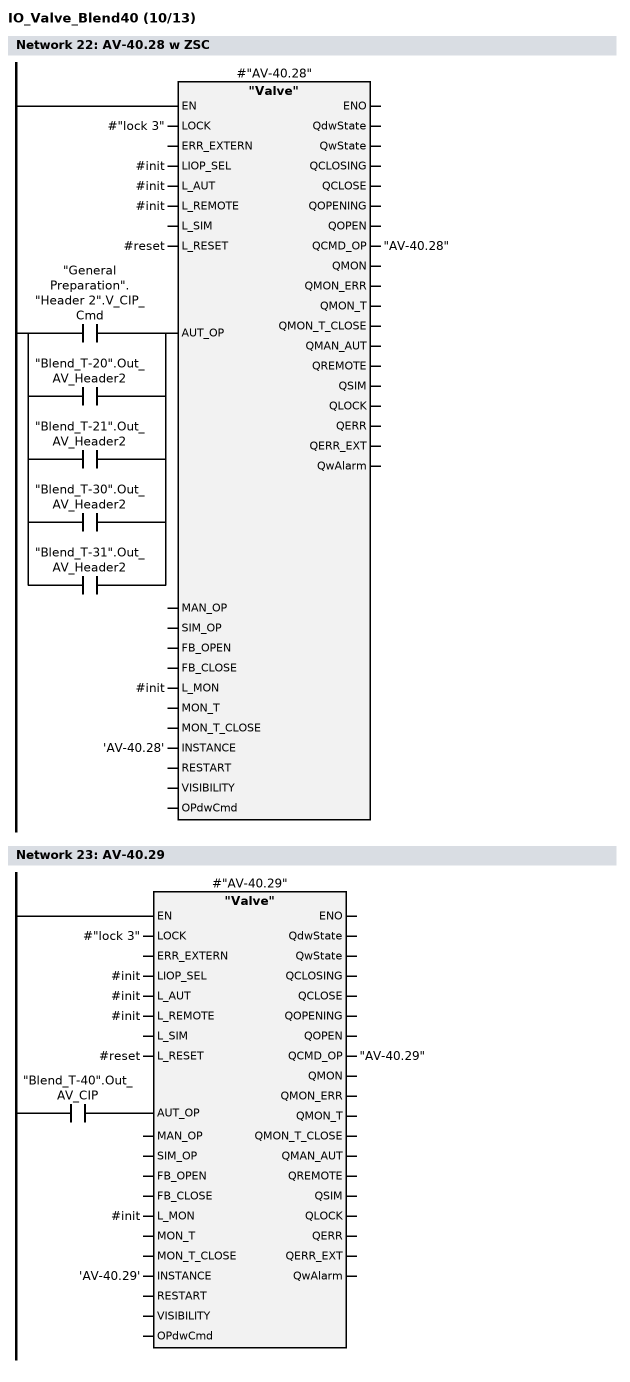
   RUNG wire#powerrail
      #"AV-40.28"(AUT_OP := wire#w1, LOCK := #"lock 3", ERR_EXTERN :=, LIOP_SEL := #init, L_AUT := #init, L_REMOTE := #init, L_SIM :=, L_RESET := #reset, MAN_OP :=, SIM_OP :=, FB_OPEN :=, FB_CLOSE :=, L_MON := #init, MON_T :=, MON_T_CLOSE :=, INSTANCE := 'AV-40.28', RESTART :=, VISIBILITY :=, OPdwCmd :=, QdwState =>, QwState =>, QCLOSING =>, QCLOSE =>, QOPENING =>, QOPEN =>, QCMD_OP => "AV-40.28", QMON =>, QMON_ERR =>, QMON_T =>, QMON_T_CLOSE =>, QMAN_AUT =>, QREMOTE =>, QSIM =>, QLOCK =>, QERR =>, QERR_EXT =>, QwAlarm =>)
   END_RUNG
   RUNG wire#powerrail
      Contact( "General Preparation"."Header 2".V_CIP_Cmd )
   END_RUNG wire#w1
   RUNG wire#powerrail
      Contact( "Blend_T-20".Out_AV_Header2 )
   END_RUNG wire#w1
   RUNG wire#powerrail
      Contact( "Blend_T-21".Out_AV_Header2 )
   END_RUNG wire#w1
   RUNG wire#powerrail
      Contact( "Blend_T-30".Out_AV_Header2 )
   END_RUNG wire#w1
   RUNG wire#powerrail
      Contact( "Blend_T-31".Out_AV_Header2 )
   END_RUNG wire#w1
   // the same network as SCL:
   #"AV-40.28"(LOCK := #"lock 3",   // "Valve"
               LIOP_SEL := #init,
               L_AUT := #init,
               L_REMOTE := #init,
               L_RESET := #reset,
               AUT_OP := "General Preparation"."Header 2".V_CIP_Cmd OR "Blend_T-20".Out_AV_Header2 OR "Blend_T-21".Out_AV_Header2 OR "Blend_T-30".Out_AV_Header2 OR "Blend_T-31".Out_AV_Header2,
               L_MON := #init,
               INSTANCE := 'AV-40.28',
               QCMD_OP => "AV-40.28");
END_REGION

REGION Network 23: AV-40.29
   RUNG wire#powerrail
      #"AV-40.29"(AUT_OP := wire#w1, LOCK := #"lock 3", ERR_EXTERN :=, LIOP_SEL := #init, L_AUT := #init, L_REMOTE := #init, L_SIM :=, L_RESET := #reset, MAN_OP :=, SIM_OP :=, FB_OPEN :=, FB_CLOSE :=, L_MON := #init, MON_T :=, MON_T_CLOSE :=, INSTANCE := 'AV-40.29', RESTART :=, VISIBILITY :=, OPdwCmd :=, QdwState =>, QwState =>, QCLOSING =>, QCLOSE =>, QOPENING =>, QOPEN =>, QCMD_OP => "AV-40.29", QMON =>, QMON_ERR =>, QMON_T =>, QMON_T_CLOSE =>, QMAN_AUT =>, QREMOTE =>, QSIM =>, QLOCK =>, QERR =>, QERR_EXT =>, QwAlarm =>)
   END_RUNG
   RUNG wire#powerrail
      Contact( "Blend_T-40".Out_AV_CIP )
   END_RUNG wire#w1
   // the same network as SCL:
   #"AV-40.29"(LOCK := #"lock 3",   // "Valve"
               LIOP_SEL := #init,
               L_AUT := #init,
               L_REMOTE := #init,
               L_RESET := #reset,
               AUT_OP := "Blend_T-40".Out_AV_CIP,
               L_MON := #init,
               INSTANCE := 'AV-40.29',
               QCMD_OP => "AV-40.29");
END_REGION

REGION Network 24: AV-40.30
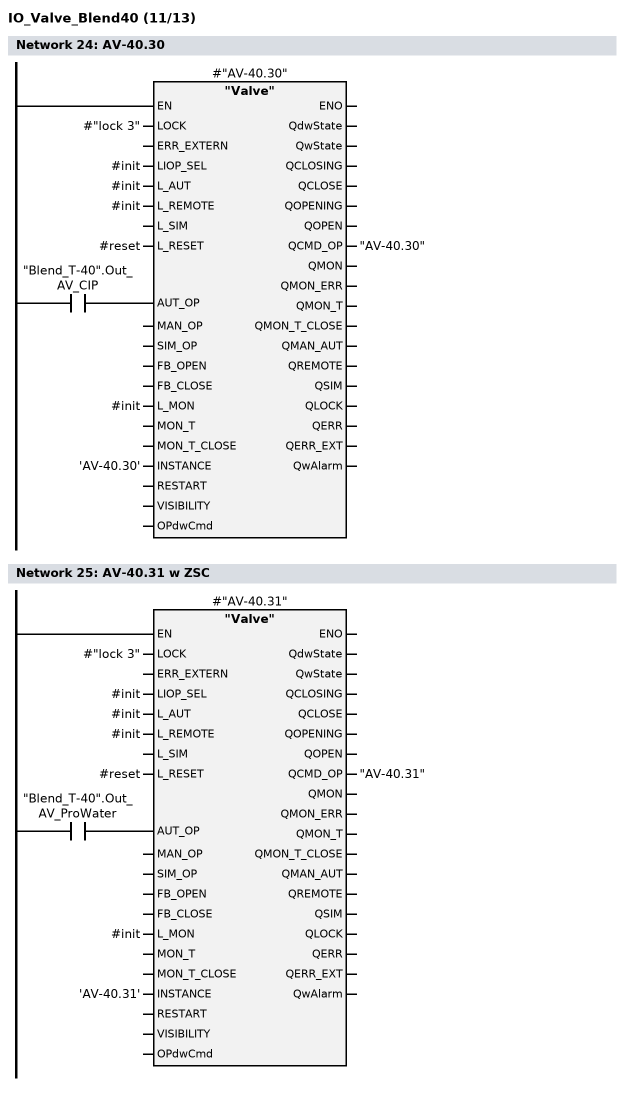
   RUNG wire#powerrail
      #"AV-40.30"(AUT_OP := wire#w1, LOCK := #"lock 3", ERR_EXTERN :=, LIOP_SEL := #init, L_AUT := #init, L_REMOTE := #init, L_SIM :=, L_RESET := #reset, MAN_OP :=, SIM_OP :=, FB_OPEN :=, FB_CLOSE :=, L_MON := #init, MON_T :=, MON_T_CLOSE :=, INSTANCE := 'AV-40.30', RESTART :=, VISIBILITY :=, OPdwCmd :=, QdwState =>, QwState =>, QCLOSING =>, QCLOSE =>, QOPENING =>, QOPEN =>, QCMD_OP => "AV-40.30", QMON =>, QMON_ERR =>, QMON_T =>, QMON_T_CLOSE =>, QMAN_AUT =>, QREMOTE =>, QSIM =>, QLOCK =>, QERR =>, QERR_EXT =>, QwAlarm =>)
   END_RUNG
   RUNG wire#powerrail
      Contact( "Blend_T-40".Out_AV_CIP )
   END_RUNG wire#w1
   // the same network as SCL:
   #"AV-40.30"(LOCK := #"lock 3",   // "Valve"
               LIOP_SEL := #init,
               L_AUT := #init,
               L_REMOTE := #init,
               L_RESET := #reset,
               AUT_OP := "Blend_T-40".Out_AV_CIP,
               L_MON := #init,
               INSTANCE := 'AV-40.30',
               QCMD_OP => "AV-40.30");
END_REGION

REGION Network 25: AV-40.31 w ZSC
   RUNG wire#powerrail
      #"AV-40.31"(AUT_OP := wire#w1, LOCK := #"lock 3", ERR_EXTERN :=, LIOP_SEL := #init, L_AUT := #init, L_REMOTE := #init, L_SIM :=, L_RESET := #reset, MAN_OP :=, SIM_OP :=, FB_OPEN :=, FB_CLOSE :=, L_MON := #init, MON_T :=, MON_T_CLOSE :=, INSTANCE := 'AV-40.31', RESTART :=, VISIBILITY :=, OPdwCmd :=, QdwState =>, QwState =>, QCLOSING =>, QCLOSE =>, QOPENING =>, QOPEN =>, QCMD_OP => "AV-40.31", QMON =>, QMON_ERR =>, QMON_T =>, QMON_T_CLOSE =>, QMAN_AUT =>, QREMOTE =>, QSIM =>, QLOCK =>, QERR =>, QERR_EXT =>, QwAlarm =>)
   END_RUNG
   RUNG wire#powerrail
      Contact( "Blend_T-40".Out_AV_ProWater )
   END_RUNG wire#w1
   // the same network as SCL:
   #"AV-40.31"(LOCK := #"lock 3",   // "Valve"
               LIOP_SEL := #init,
               L_AUT := #init,
               L_REMOTE := #init,
               L_RESET := #reset,
               AUT_OP := "Blend_T-40".Out_AV_ProWater,
               L_MON := #init,
               INSTANCE := 'AV-40.31',
               QCMD_OP => "AV-40.31");
END_REGION

REGION Network 26: AV-40.32 w ZSC
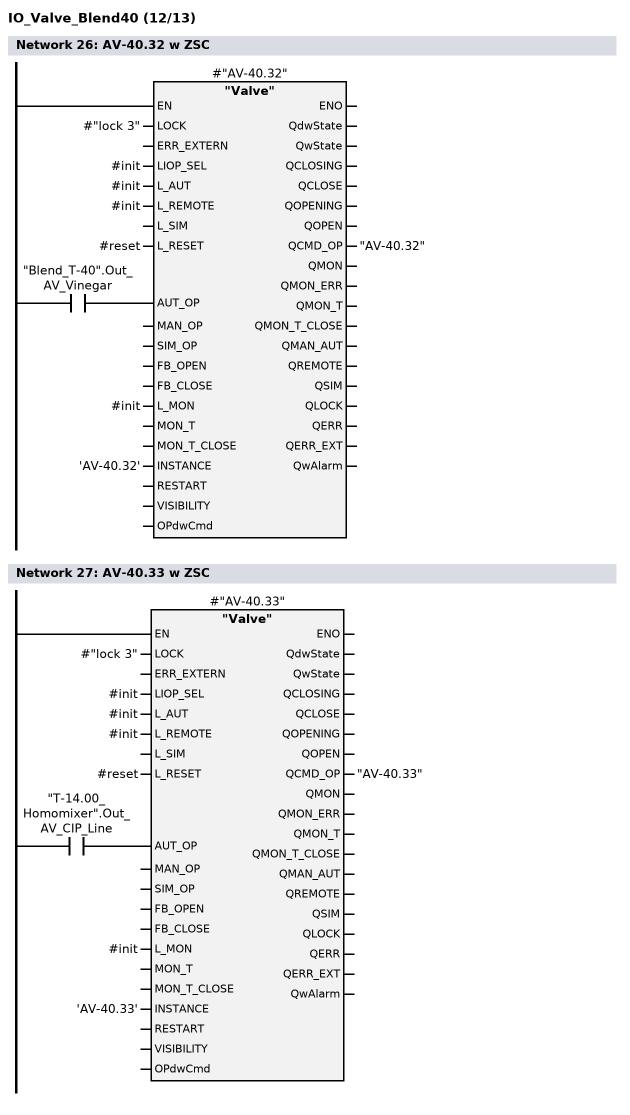
   RUNG wire#powerrail
      #"AV-40.32"(AUT_OP := wire#w1, LOCK := #"lock 3", ERR_EXTERN :=, LIOP_SEL := #init, L_AUT := #init, L_REMOTE := #init, L_SIM :=, L_RESET := #reset, MAN_OP :=, SIM_OP :=, FB_OPEN :=, FB_CLOSE :=, L_MON := #init, MON_T :=, MON_T_CLOSE :=, INSTANCE := 'AV-40.32', RESTART :=, VISIBILITY :=, OPdwCmd :=, QdwState =>, QwState =>, QCLOSING =>, QCLOSE =>, QOPENING =>, QOPEN =>, QCMD_OP => "AV-40.32", QMON =>, QMON_ERR =>, QMON_T =>, QMON_T_CLOSE =>, QMAN_AUT =>, QREMOTE =>, QSIM =>, QLOCK =>, QERR =>, QERR_EXT =>, QwAlarm =>)
   END_RUNG
   RUNG wire#powerrail
      Contact( "Blend_T-40".Out_AV_Vinegar )
   END_RUNG wire#w1
   // the same network as SCL:
   #"AV-40.32"(LOCK := #"lock 3",   // "Valve"
               LIOP_SEL := #init,
               L_AUT := #init,
               L_REMOTE := #init,
               L_RESET := #reset,
               AUT_OP := "Blend_T-40".Out_AV_Vinegar,
               L_MON := #init,
               INSTANCE := 'AV-40.32',
               QCMD_OP => "AV-40.32");
END_REGION

REGION Network 27: AV-40.33 w ZSC
   RUNG wire#powerrail
      #"AV-40.33"(AUT_OP := wire#w1, LOCK := #"lock 3", ERR_EXTERN :=, LIOP_SEL := #init, L_AUT := #init, L_REMOTE := #init, L_SIM :=, L_RESET := #reset, MAN_OP :=, SIM_OP :=, FB_OPEN :=, FB_CLOSE :=, L_MON := #init, MON_T :=, MON_T_CLOSE :=, INSTANCE := 'AV-40.33', RESTART :=, VISIBILITY :=, OPdwCmd :=, QdwState =>, QwState =>, QCLOSING =>, QCLOSE =>, QOPENING =>, QOPEN =>, QCMD_OP => "AV-40.33", QMON =>, QMON_ERR =>, QMON_T =>, QMON_T_CLOSE =>, QMAN_AUT =>, QREMOTE =>, QSIM =>, QLOCK =>, QERR =>, QERR_EXT =>, QwAlarm =>)
   END_RUNG
   RUNG wire#powerrail
      Contact( "T-14.00_Homomixer".Out_AV_CIP_Line )
   END_RUNG wire#w1
   // the same network as SCL:
   #"AV-40.33"(LOCK := #"lock 3",   // "Valve"
               LIOP_SEL := #init,
               L_AUT := #init,
               L_REMOTE := #init,
               L_RESET := #reset,
               AUT_OP := "T-14.00_Homomixer".Out_AV_CIP_Line,
               L_MON := #init,
               INSTANCE := 'AV-40.33',
               QCMD_OP => "AV-40.33");
END_REGION

REGION Network 28: AV-40.34 w ZSC
